KUKA KRL program: MyProgram_175().src

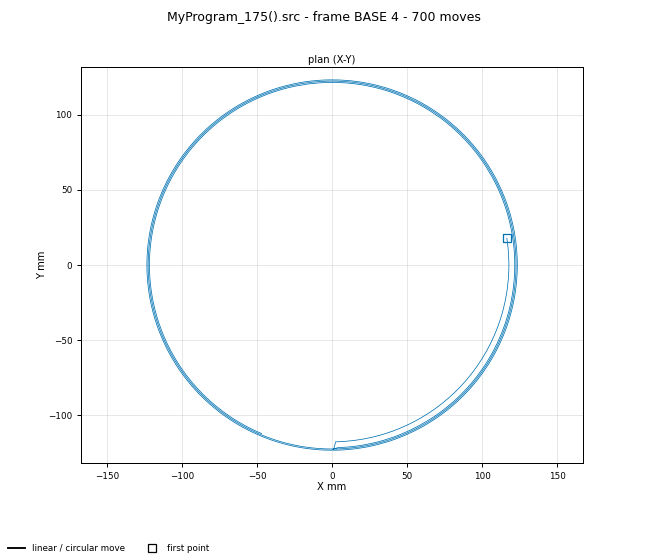
[picture p0: tool path of MyProgram_175().src in frame BASE 4, 700 of 700 moves have a stored position in this frame; points joined in program order, loops and branches not executed]
&ACCESS RVP
&REL 1
&PARAM TEMPLATE = C:\KRC\Roboter\Template\vorgabe
&PARAM EDITMASK = *
DEF MyProgram_175()
; ---- Setting reference (Base) ----
$BASE = BASE_DATA[4]

; --------------------------
; ---- Setting tool (TCP) ----
$TOOL = TOOL_DATA[3]
; --------------------------

$VEL.CP = VEL_APROX_PRINT
Startdeposition()
$VEL.CP = VEL_PRINT
LIN {X 116.3937,Y 17.9256,Z 129,A 4.4321,B 24.9467,C -1.6867,E1 25.1581,E2 441.6047} C_DIS
LIN {X 116.7972,Y 15.0743,Z 129,A 3.0217,B 24.947,C -1.6817,E1 25.1586,E2 443.0185} C_DIS
LIN {X 117.1569,Y 11.9651,Z 129,A 1.4665,B 24.9474,C -1.6752,E1 25.1591,E2 444.5798} C_DIS
LIN {X 117.4486,Y 8.67,Z 129,A -0.1015,B 24.9476,C -1.672,E1 25.1594,E2 446.1462} C_DIS
LIN {X 117.6272,Y 5.7574,Z 129,A -1.4975,B 24.9478,C -1.6685,E1 25.1596,E2 447.5421} C_DIS
LIN {X 117.7329,Y 2.8788,Z 129,A -2.8893,B 24.9481,C -1.6644,E1 25.1598,E2 448.9353} C_DIS
LIN {X 117.7651,Y -0.5226,Z 129,A -4.5792,B 24.9485,C -1.6573,E1 25.1598,E2 450.6318} C_DIS
LIN {X 117.7122,Y -3.559,Z 129,A -6.025,B 24.9487,C -1.654,E1 25.1597,E2 452.0768} C_DIS
LIN {X 117.5839,Y -6.5462,Z 129,A -7.4486,B 24.9489,C -1.6507,E1 25.1595,E2 453.4997} C_DIS
LIN {X 117.394,Y -9.3527,Z 129,A -8.8238,B 24.9492,C -1.6459,E1 25.1592,E2 454.8781} C_DIS
LIN {X 117.1208,Y -12.3096,Z 129,A -10.2202,B 24.9494,C -1.6435,E1 25.1588,E2 456.2718} C_DIS
LIN {X 116.796,Y -15.0832,Z 129,A -11.6081,B 24.9497,C -1.6377,E1 25.1583,E2 457.6654} C_DIS
LIN {X 116.3879,Y -17.9631,Z 129,A -13.0134,B 24.95,C -1.6335,E1 25.1578,E2 459.0722} C_DIS
LIN {X 115.8974,Y -20.8952,Z 129,A -14.4115,B 24.9501,C -1.6311,E1 25.1571,E2 460.4677} C_DIS
LIN {X 115.3444,Y -23.759,Z 129,A -15.8145,B 24.9504,C -1.6273,E1 25.1563,E2 461.8716} C_DIS
LIN {X 114.7348,Y -26.5469,Z 129,A -17.1994,B 24.9506,C -1.623,E1 25.1555,E2 463.2586} C_DIS
LIN {X 114.0503,Y -29.3488,Z 129,A -18.6126,B 24.9509,C -1.6179,E1 25.1545,E2 464.6755} C_DIS
LIN {X 113.3216,Y -32.0474,Z 129,A -20.0108,B 24.9513,C -1.6117,E1 25.1535,E2 466.0803} C_DIS
LIN {X 112.2615,Y -35.59,Z 129,A -21.7488,B 24.9515,C -1.6089,E1 25.1521,E2 467.8151} C_DIS
LIN {X 111.3572,Y -38.326,Z 129,A -23.1413,B 24.9517,C -1.6049,E1 25.1508,E2 469.2092} C_DIS
LIN {X 110.3859,Y -41.0399,Z 129,A -24.5345,B 24.952,C -1.6009,E1 25.1495,E2 470.6039} C_DIS
LIN {X 109.1507,Y -44.2152,Z 129,A -26.2203,B 24.9524,C -1.5944,E1 25.1478,E2 472.2957} C_DIS
LIN {X 107.975,Y -47.013,Z 129,A -27.6487,B 24.9525,C -1.5922,E1 25.1462,E2 473.7217} C_DIS
LIN {X 106.7548,Y -49.7216,Z 129,A -29.0647,B 24.9527,C -1.5891,E1 25.1445,E2 475.1371} C_DIS
LIN {X 105.5449,Y -52.2407,Z 129,A -30.4738,B 24.9531,C -1.5826,E1 25.1428,E2 476.5539} C_DIS
LIN {X 104.167,Y -54.9368,Z 129,A -31.8799,B 24.9531,C -1.5814,E1 25.141,E2 477.9555} C_DIS
LIN {X 102.7942,Y -57.4645,Z 129,A -33.2704,B 24.9534,C -1.5777,E1 25.1391,E2 479.3475} C_DIS
LIN {X 101.4046,Y -59.8827,Z 129,A -34.6519,B 24.9537,C -1.5725,E1 25.1372,E2 480.7341} C_DIS
LIN {X 99.8534,Y -62.4349,Z 129,A -36.083,B 24.9539,C -1.5693,E1 25.1351,E2 482.1655} C_DIS
LIN {X 98.3422,Y -64.7891,Z 129,A -37.4354,B 24.9541,C -1.5658,E1 25.133,E2 483.5193} C_DIS
LIN {X 96.7259,Y -67.1783,Z 129,A -38.8304,B 24.9543,C -1.5623,E1 25.1308,E2 484.9158} C_DIS
LIN {X 95.0339,Y -69.5512,Z 129,A -40.2395,B 24.9545,C -1.5587,E1 25.1285,E2 486.3264} C_DIS
LIN {X 93.2787,Y -71.8881,Z 129,A -41.6535,B 24.9547,C -1.5552,E1 25.1261,E2 487.742} C_DIS
LIN {X 91.4909,Y -74.1501,Z 129,A -43.0481,B 24.9549,C -1.5518,E1 25.1237,E2 489.1381} C_DIS
LIN {X 89.6483,Y -76.3676,Z 129,A -44.4513,B 24.9551,C -1.5481,E1 25.1212,E2 490.5437} C_DIS
LIN {X 87.728,Y -78.566,Z 129,A -45.8549,B 24.9553,C -1.5452,E1 25.1186,E2 491.9479} C_DIS
LIN {X 85.7806,Y -80.6877,Z 129,A -47.2487,B 24.9555,C -1.5419,E1 25.1159,E2 493.3432} C_DIS
LIN {X 83.7811,Y -82.7619,Z 129,A -48.6429,B 24.9556,C -1.5388,E1 25.1132,E2 494.7389} C_DIS
LIN {X 81.7314,Y -84.7867,Z 129,A -50.0452,B 24.9558,C -1.5353,E1 25.1104,E2 496.1434} C_DIS
LIN {X 79.6064,Y -86.785,Z 129,A -51.4495,B 24.956,C -1.5326,E1 25.1075,E2 497.5483} C_DIS
LIN {X 77.4591,Y -88.7069,Z 129,A -52.8446,B 24.9562,C -1.5297,E1 25.1046,E2 498.9449} C_DIS
LIN {X 75.2647,Y -90.5761,Z 129,A -54.2403,B 24.9563,C -1.5268,E1 25.1016,E2 500.3421} C_DIS
LIN {X 73.0251,Y -92.3913,Z 129,A -55.6361,B 24.9565,C -1.524,E1 25.0986,E2 501.7393} C_DIS
LIN {X 70.7095,Y -94.1753,Z 129,A -57.0586,B 24.9567,C -1.5209,E1 25.0954,E2 503.1639} C_DIS
LIN {X 68.3563,Y -95.897,Z 129,A -58.4643,B 24.9567,C -1.5185,E1 25.0922,E2 504.5702} C_DIS
LIN {X 65.9875,Y -97.5422,Z 129,A -59.8614,B 24.9569,C -1.516,E1 25.089,E2 505.9686} C_DIS
LIN {X 63.6275,Y -99.0977,Z 129,A -61.2294,B 24.9571,C -1.5136,E1 25.0858,E2 507.3377} C_DIS
LIN {X 61.1156,Y -100.6663,Z 129,A -62.6648,B 24.9572,C -1.5111,E1 25.0824,E2 508.7746} C_DIS
LIN {X 58.6405,Y -102.1279,Z 129,A -64.0379,B 24.9573,C -1.5097,E1 25.0791,E2 510.1468} C_DIS
LIN {X 56.131,Y -103.5284,Z 129,A -65.4376,B 24.9574,C -1.5071,E1 25.0756,E2 511.5484} C_DIS
LIN {X 53.4791,Y -104.9229,Z 129,A -66.8953,B 24.9576,C -1.5046,E1 25.072,E2 513.008} C_DIS
LIN {X 50.9395,Y -106.1791,Z 129,A -68.2585,B 24.9576,C -1.5031,E1 25.0686,E2 514.3712} C_DIS
LIN {X 48.3281,Y -107.3928,Z 129,A -69.6738,B 24.9578,C -1.5002,E1 25.065,E2 515.7897} C_DIS
LIN {X 45.6867,Y -108.5428,Z 129,A -71.0517,B 24.9578,C -1.4992,E1 25.0615,E2 517.1667} C_DIS
LIN {X 43.0999,Y -109.5957,Z 129,A -72.4452,B 24.9581,C -1.4956,E1 25.0578,E2 518.5655} C_DIS
LIN {X 40.3227,Y -110.6476,Z 129,A -73.8663,B 24.9581,C -1.4948,E1 25.0541,E2 519.9856} C_DIS
LIN {X 37.6045,Y -111.6007,Z 129,A -75.2508,B 24.9581,C -1.4938,E1 25.0505,E2 521.3698} C_DIS
LIN {X 34.8327,Y -112.4967,Z 129,A -76.7077,B 24.9584,C -1.4902,E1 25.0466,E2 522.8324} C_DIS
LIN {X 31.3934,Y -113.5067,Z 129,A -78.4167,B 24.9584,C -1.4898,E1 25.042,E2 524.5395} C_DIS
LIN {X 28.6049,Y -114.2414,Z 129,A -79.8167,B 24.9584,C -1.4885,E1 25.0382,E2 525.9405} C_DIS
LIN {X 25.7987,Y -114.9076,Z 129,A -81.2172,B 24.9586,C -1.4873,E1 25.0344,E2 527.342} C_DIS
LIN {X 22.9256,Y -115.5149,Z 129,A -82.6405,B 24.9586,C -1.4863,E1 25.0305,E2 528.7659} C_DIS
LIN {X 20.1009,Y -116.0398,Z 129,A -84.0367,B 24.9586,C -1.4852,E1 25.0267,E2 530.163} C_DIS
LIN {X 17.2609,Y -116.4962,Z 129,A -85.4392,B 24.9587,C -1.484,E1 25.0228,E2 531.567} C_DIS
LIN {X 14.409,Y -116.8833,Z 129,A -86.8328,B 24.9587,C -1.4834,E1 25.0189,E2 532.9609} C_DIS
LIN {X 11.5196,Y -117.2033,Z 129,A -88.2452,B 24.9588,C -1.4827,E1 25.015,E2 534.374} C_DIS
LIN {X 8.653,Y -117.4498,Z 129,A -89.7448,B 24.9591,C -1.4775,E1 25.0108,E2 535.8853} C_DIS
LIN {X 5.7539,Y -117.6274,Z 129,A -91.0554,B 24.9589,C -1.4815,E1 25.0072,E2 537.1858} C_DIS
LIN {X 2.394,Y -117.7418,Z 129,A -92.7403,B 24.959,C -1.4788,E1 25.0024,E2 538.8768} C_DIS
LIN {X 2.394,Y -117.7418,Z 129,A -92.7403,B 24.959,C -1.4788,E1 25.0024,E2 538.8768} C_DIS
Enddeposition()
LIN {X 0.876,Y -123.3662,Z 130,A -92.9891,B 24.9627,C -1.4112,E1 25.0013,E2 539.2857} C_DIS
Startdeposition()
$VEL.CP = VEL_PRINT
LIN {X 3.429,Y -123.3221,Z 130,A -91.439,B 24.9617,C -1.4291,E1 25.0058,E2 537.6935} C_DIS
LIN {X 6.0536,Y -123.2229,Z 130,A -90.0878,B 24.9614,C -1.4359,E1 25.0096,E2 536.3266} C_DIS
LIN {X 9.4299,Y -123.0089,Z 130,A -88.6359,B 24.9616,C -1.4309,E1 25.0136,E2 534.8873} C_DIS
LIN {X 12.4918,Y -122.7357,Z 130,A -87.2244,B 24.9616,C -1.4309,E1 25.0175,E2 533.4767} C_DIS
LIN {X 15.102,Y -122.4437,Z 130,A -86.0061,B 24.9616,C -1.4315,E1 25.0209,E2 532.2577} C_DIS
LIN {X 18.4991,Y -121.9749,Z 130,A -84.4157,B 24.9616,C -1.4325,E1 25.0253,E2 530.6664} C_DIS
LIN {X 21.0918,Y -121.5552,Z 130,A -83.0658,B 24.9612,C -1.4398,E1 25.029,E2 529.3006} C_DIS
LIN {X 24.0686,Y -121.001,Z 130,A -81.6622,B 24.9612,C -1.4409,E1 25.0329,E2 527.8961} C_DIS
LIN {X 27.422,Y -120.2835,Z 130,A -80.2048,B 24.9614,C -1.4358,E1 25.0368,E2 526.4527} C_DIS
LIN {X 29.9768,Y -119.6742,Z 130,A -78.9876,B 24.9614,C -1.4368,E1 25.0401,E2 525.2348} C_DIS
LIN {X 33.291,Y -118.7931,Z 130,A -77.5658,B 24.9617,C -1.4302,E1 25.0439,E2 523.831} C_DIS
LIN {X 35.8129,Y -118.0592,Z 130,A -76.1817,B 24.9612,C -1.4397,E1 25.0477,E2 522.4269} C_DIS
LIN {X 38.6994,Y -117.1447,Z 130,A -74.7791,B 24.9611,C -1.4412,E1 25.0514,E2 521.0233} C_DIS
LIN {X 41.5626,Y -116.1597,Z 130,A -73.3767,B 24.9611,C -1.4429,E1 25.0551,E2 519.6198} C_DIS
LIN {X 44.7745,Y -114.958,Z 130,A -71.784,B 24.9609,C -1.4451,E1 25.0592,E2 518.0252} C_DIS
LIN {X 47.2122,Y -113.9804,Z 130,A -70.5726,B 24.9609,C -1.4464,E1 25.0624,E2 516.8135} C_DIS
LIN {X 50.3612,Y -112.6225,Z 130,A -68.9852,B 24.9607,C -1.4486,E1 25.0664,E2 515.2248} C_DIS
LIN {X 53.11,Y -111.3527,Z 130,A -67.7507,B 24.961,C -1.4424,E1 25.0695,E2 514.0082} C_DIS
LIN {X 55.4692,Y -110.1985,Z 130,A -66.2126,B 24.9601,C -1.4602,E1 25.0735,E2 512.4322} C_DIS
LIN {X 58.5098,Y -108.6126,Z 130,A -64.7813,B 24.9603,C -1.455,E1 25.0769,E2 511.0173} C_DIS
LIN {X 61.1577,Y -107.144,Z 130,A -63.5474,B 24.9607,C -1.4489,E1 25.0799,E2 509.8014} C_DIS
LIN {X 63.7687,Y -105.6108,Z 130,A -62.0577,B 24.9603,C -1.4557,E1 25.0835,E2 508.3002} C_DIS
LIN {X 66.3413,Y -104.014,Z 130,A -60.5698,B 24.9599,C -1.4625,E1 25.0871,E2 506.8009} C_DIS
LIN {X 68.601,Y -102.5394,Z 130,A -59.3612,B 24.9599,C -1.4628,E1 25.0899,E2 505.5958} C_DIS
LIN {X 71.0383,Y -100.8667,Z 130,A -57.9646,B 24.9597,C -1.4668,E1 25.0931,E2 504.1945} C_DIS
LIN {X 73.8133,Y -98.8518,Z 130,A -56.3792,B 24.9595,C -1.4698,E1 25.0966,E2 502.6075} C_DIS
LIN {X 75.9021,Y -97.2595,Z 130,A -55.0333,B 24.959,C -1.4788,E1 25.0997,E2 501.2453} C_DIS
LIN {X 78.2661,Y -95.3675,Z 130,A -53.6536,B 24.959,C -1.4806,E1 25.1026,E2 499.8665} C_DIS
LIN {X 80.5829,Y -93.418,Z 130,A -52.2344,B 24.9587,C -1.4845,E1 25.1057,E2 498.4437} C_DIS
LIN {X 83.1471,Y -91.1409,Z 130,A -50.9478,B 24.9594,C -1.4729,E1 25.1083,E2 497.1898} C_DIS
LIN {X 85.0697,Y -89.3515,Z 130,A -49.4363,B 24.9584,C -1.4905,E1 25.1114,E2 495.6428} C_DIS
LIN {X 87.2368,Y -87.2368,Z 130,A -48.0373,B 24.9582,C -1.4936,E1 25.1142,E2 494.2424} C_DIS
LIN {X 89.6265,Y -84.7772,Z 130,A -46.7511,B 24.9588,C -1.4822,E1 25.1166,E2 492.9888} C_DIS
LIN {X 91.4123,Y -82.8513,Z 130,A -45.2399,B 24.9578,C -1.5001,E1 25.1195,E2 491.4421} C_DIS
LIN {X 93.6784,Y -80.2773,Z 130,A -43.7876,B 24.958,C -1.4971,E1 25.1222,E2 490.0032} C_DIS
LIN {X 95.3675,Y -78.2661,Z 130,A -42.443,B 24.9575,C -1.5067,E1 25.1246,E2 488.6423} C_DIS
LIN {X 97.2595,Y -75.9021,Z 130,A -41.1765,B 24.9577,C -1.5034,E1 25.1267,E2 487.3895} C_DIS
LIN {X 99.3301,Y -73.1684,Z 130,A -39.5931,B 24.9574,C -1.5074,E1 25.1294,E2 485.8044} C_DIS
LIN {X 101.0958,Y -70.7087,Z 130,A -38.1953,B 24.9572,C -1.5109,E1 25.1316,E2 484.4051} C_DIS
LIN {X 102.8755,Y -68.0929,Z 130,A -36.9573,B 24.9577,C -1.5033,E1 25.1335,E2 483.191} C_DIS
LIN {X 104.4436,Y -65.663,Z 130,A -35.5665,B 24.9573,C -1.5096,E1 25.1357,E2 481.7924} C_DIS
LIN {X 106.0236,Y -63.0801,Z 130,A -34.1685,B 24.9571,C -1.5132,E1 25.1377,E2 480.3929} C_DIS
LIN {X 107.344,Y -60.8096,Z 130,A -32.79,B 24.9564,C -1.5249,E1 25.1396,E2 478.994} C_DIS
LIN {X 108.991,Y -57.8017,Z 130,A -31.2074,B 24.9562,C -1.5292,E1 25.1417,E2 477.4096} C_DIS
LIN {X 110.3767,Y -55.1096,Z 130,A -29.9764,B 24.9565,C -1.5245,E1 25.1433,E2 476.1962} C_DIS
LIN {X 111.5265,Y -52.7481,Z 130,A -28.5983,B 24.9558,C -1.5363,E1 25.1449,E2 474.7977} C_DIS
LIN {X 112.9479,Y -49.6272,Z 130,A -27.0159,B 24.9555,C -1.5407,E1 25.1468,E2 473.2135} C_DIS
LIN {X 113.9804,Y -47.2122,Z 130,A -25.8038,B 24.9553,C -1.5441,E1 25.1481,E2 472.0002} C_DIS
LIN {X 115.2469,Y -44.0254,Z 130,A -24.177,B 24.9549,C -1.5509,E1 25.1497,E2 470.3665} C_DIS
LIN {X 116.2927,Y -41.1838,Z 130,A -22.825,B 24.9549,C -1.5525,E1 25.151,E2 469.0181} C_DIS
LIN {X 117.2683,Y -38.3174,Z 130,A -21.4284,B 24.9546,C -1.5565,E1 25.1522,E2 467.62} C_DIS
LIN {X 118.1734,Y -35.428,Z 130,A -20.1978,B 24.9549,C -1.552,E1 25.1532,E2 466.407} C_DIS
LIN {X 119.0072,Y -32.5172,Z 130,A -18.6351,B 24.9541,C -1.5645,E1 25.1544,E2 464.8237} C_DIS
LIN {X 119.6742,Y -29.9768,Z 130,A -17.3374,B 24.9537,C -1.5724,E1 25.1553,E2 463.5149} C_DIS
LIN {X 120.4667,Y -26.6053,Z 130,A -15.8289,B 24.9537,C -1.5726,E1 25.1563,E2 462.0148} C_DIS
LIN {X 121.001,Y -24.0686,Z 130,A -14.4988,B 24.9531,C -1.5829,E1 25.157,E2 460.6681} C_DIS
LIN {X 121.5552,Y -21.0918,Z 130,A -13.2337,B 24.9532,C -1.5803,E1 25.1576,E2 459.4166} C_DIS
LIN {X 122.0927,Y -17.7049,Z 130,A -11.6521,B 24.9529,C -1.5849,E1 25.1583,E2 457.8334} C_DIS
LIN {X 122.6198,Y -13.5983,Z 130,A -9.7423,B 24.9526,C -1.5905,E1 25.1589,E2 455.9216} C_DIS
LIN {X 122.9486,Y -10.1848,Z 130,A -8.3272,B 24.9528,C -1.5867,E1 25.1593,E2 454.5239} C_DIS
LIN {X 123.1615,Y -7.1644,Z 130,A -6.9306,B 24.9526,C -1.5908,E1 25.1596,E2 453.1259} C_DIS
LIN {X 123.2879,Y -4.541,Z 130,A -5.4214,B 24.9515,C -1.6097,E1 25.1597,E2 451.5813} C_DIS
LIN {X 123.3622,Y -1.514,Z 130,A -4.0379,B 24.9512,C -1.6131,E1 25.1597,E2 450.198} C_DIS
LIN {X 123.3607,Y 1.5958,Z 130,A -2.6187,B 24.951,C -1.6165,E1 25.1597,E2 448.779} C_DIS
LIN {X 123.2707,Y 4.942,Z 130,A -1.3446,B 24.9516,C -1.6073,E1 25.1597,E2 447.5344} C_DIS
LIN {X 123.1123,Y 7.9658,Z 130,A 0.0521,B 24.9513,C -1.6114,E1 25.1594,E2 446.1363} C_DIS
LIN {X 122.9166,Y 10.5849,Z 130,A 1.5614,B 24.9502,C -1.6301,E1 25.1591,E2 444.5918} C_DIS
LIN {X 122.5731,Y 13.997,Z 130,A 3.0115,B 24.9503,C -1.628,E1 25.1586,E2 443.1553} C_DIS
LIN {X 122.1927,Y 17.0009,Z 130,A 4.4082,B 24.9501,C -1.632,E1 25.1581,E2 441.7573} C_DIS
LIN {X 121.7387,Y 19.9945,Z 130,A 5.6386,B 24.9504,C -1.6276,E1 25.1576,E2 440.5446} C_DIS
LIN {X 121.2113,Y 22.9761,Z 130,A 7.2015,B 24.9496,C -1.64,E1 25.1568,E2 438.9615} C_DIS
LIN {X 120.611,Y 25.9439,Z 130,A 8.6253,B 24.9493,C -1.6454,E1 25.156,E2 437.5334} C_DIS
LIN {X 119.6742,Y 29.9768,Z 130,A 10.5089,B 24.949,C -1.6494,E1 25.1548,E2 435.6512} C_DIS
LIN {X 118.9025,Y 32.9048,Z 130,A 11.9058,B 24.9488,C -1.6533,E1 25.1537,E2 434.2532} C_DIS
LIN {X 118.0592,Y 35.8129,Z 130,A 13.3029,B 24.9485,C -1.6572,E1 25.1526,E2 432.855} C_DIS
LIN {X 117.1448,Y 38.6994,Z 130,A 14.8315,B 24.9479,C -1.6677,E1 25.1513,E2 431.3101} C_DIS
LIN {X 116.1597,Y 41.5626,Z 130,A 16.0973,B 24.9481,C -1.6648,E1 25.1501,E2 430.0584} C_DIS
LIN {X 115.1048,Y 44.4008,Z 130,A 17.5072,B 24.9478,C -1.6692,E1 25.1487,E2 428.6459} C_DIS
LIN {X 113.8245,Y 47.5822,Z 130,A 18.911,B 24.9481,C -1.6643,E1 25.1473,E2 427.2613} C_DIS
LIN {X 112.7875,Y 49.9952,Z 130,A 20.3887,B 24.9471,C -1.6809,E1 25.1456,E2 425.7526} C_DIS
LIN {X 111.3527,Y 53.11,Z 130,A 21.7062,B 24.9476,C -1.6716,E1 25.1441,E2 424.4641} C_DIS
LIN {X 110.1985,Y 55.4692,Z 130,A 23.0851,B 24.9469,C -1.6831,E1 25.1423,E2 423.0655} C_DIS
LIN {X 108.6126,Y 58.5098,Z 130,A 24.6684,B 24.9467,C -1.6871,E1 25.1403,E2 421.4811} C_DIS
LIN {X 107.144,Y 61.1577,Z 130,A 26.0664,B 24.9464,C -1.6906,E1 25.1383,E2 420.0822} C_DIS
LIN {X 105.6108,Y 63.7687,Z 130,A 27.2981,B 24.9468,C -1.6856,E1 25.1366,E2 418.8686} C_DIS
LIN {X 104.2309,Y 66.0035,Z 130,A 28.7053,B 24.946,C -1.6982,E1 25.1345,E2 417.4386} C_DIS
LIN {X 102.3546,Y 68.874,Z 130,A 30.0946,B 24.9463,C -1.6922,E1 25.1324,E2 416.0704} C_DIS
LIN {X 100.6335,Y 71.3651,Z 130,A 31.6599,B 24.9456,C -1.7038,E1 25.1299,E2 414.4854} C_DIS
LIN {X 98.8518,Y 73.8133,Z 130,A 33.0587,B 24.9454,C -1.707,E1 25.1275,E2 413.0859} C_DIS
LIN {X 97.0106,Y 76.217,Z 130,A 34.2907,B 24.9457,C -1.7017,E1 25.1255,E2 411.8721} C_DIS
LIN {X 95.1109,Y 78.5748,Z 130,A 35.6897,B 24.9455,C -1.7047,E1 25.123,E2 410.4725} C_DIS
LIN {X 93.418,Y 80.5829,Z 130,A 37.0705,B 24.9448,C -1.7156,E1 25.1205,E2 409.0724} C_DIS
LIN {X 91.4123,Y 82.8513,Z 130,A 38.4701,B 24.9447,C -1.7185,E1 25.1179,E2 407.6721} C_DIS
LIN {X 89.0729,Y 85.3587,Z 130,A 39.888,B 24.945,C -1.7134,E1 25.1152,E2 406.2724} C_DIS
LIN {X 86.9512,Y 87.519,Z 130,A 41.4546,B 24.9443,C -1.7245,E1 25.1121,E2 404.6864} C_DIS
LIN {X 84.7772,Y 89.6265,Z 130,A 42.6878,B 24.9446,C -1.7189,E1 25.1096,E2 403.4715} C_DIS
LIN {X 82.8513,Y 91.4123,Z 130,A 44.0692,B 24.944,C -1.7294,E1 25.1067,E2 402.071} C_DIS
LIN {X 80.3955,Y 93.5777,Z 130,A 45.5306,B 24.944,C -1.7295,E1 25.1037,E2 400.615} C_DIS
LIN {X 78.2661,Y 95.3675,Z 130,A 46.87,B 24.9436,C -1.7343,E1 25.1008,E2 399.2693} C_DIS
LIN {X 75.5841,Y 97.5045,Z 130,A 48.4562,B 24.9435,C -1.737,E1 25.0973,E2 397.6826} C_DIS
LIN {X 73.1684,Y 99.3301,Z 130,A 49.6903,B 24.9438,C -1.7311,E1 25.0946,E2 396.467} C_DIS
LIN {X 71.0383,Y 100.8667,Z 130,A 51.2044,B 24.9428,C -1.7477,E1 25.0911,E2 394.919} C_DIS
LIN {X 68.2064,Y 102.8007,Z 130,A 52.6595,B 24.943,C -1.7436,E1 25.0877,E2 393.4785} C_DIS
LIN {X 66.0035,Y 104.2309,Z 130,A 54.0337,B 24.9424,C -1.7531,E1 25.0844,E2 392.0863} C_DIS
LIN {X 63.0801,Y 106.0236,Z 130,A 55.2956,B 24.9433,C -1.7393,E1 25.0815,E2 390.8609} C_DIS
LIN {X 60.8096,Y 107.344,Z 130,A 56.8108,B 24.9422,C -1.7555,E1 25.0778,E2 389.312} C_DIS
LIN {X 57.8017,Y 108.991,Z 130,A 58.0995,B 24.9431,C -1.7429,E1 25.0747,E2 388.0567} C_DIS
LIN {X 55.1096,Y 110.3767,Z 130,A 59.6689,B 24.9424,C -1.7527,E1 25.0707,E2 386.4685} C_DIS
LIN {X 52.3842,Y 111.696,Z 130,A 60.9044,B 24.9429,C -1.7461,E1 25.0676,E2 385.2518} C_DIS
LIN {X 49.9952,Y 112.7875,Z 130,A 62.2885,B 24.9422,C -1.7555,E1 25.0641,E2 383.8489} C_DIS
LIN {X 47.2122,Y 113.9804,Z 130,A 63.6918,B 24.9422,C -1.7568,E1 25.0605,E2 382.4457} C_DIS
LIN {X 44.4008,Y 115.1048,Z 130,A 65.0947,B 24.9421,C -1.7581,E1 25.0568,E2 381.0429} C_DIS
LIN {X 41.5081,Y 116.1789,Z 130,A 66.5008,B 24.9421,C -1.7581,E1 25.0531,E2 379.6396} C_DIS
LIN {X 38.6994,Y 117.1447,Z 130,A 67.9019,B 24.9419,C -1.7604,E1 25.0494,E2 378.236} C_DIS
LIN {X 35.428,Y 118.1734,Z 130,A 69.4918,B 24.9419,C -1.7615,E1 25.0452,E2 376.6463} C_DIS
LIN {X 32.5172,Y 119.0072,Z 130,A 70.7285,B 24.9423,C -1.7543,E1 25.0419,E2 375.4285} C_DIS
LIN {X 29.9768,Y 119.6742,Z 130,A 72.2466,B 24.9413,C -1.7694,E1 25.0377,E2 373.8771} C_DIS
LIN {X 27.0309,Y 120.3739,Z 130,A 73.6515,B 24.9413,C -1.7701,E1 25.0339,E2 372.4726} C_DIS
LIN {X 24.0686,Y 121.001,Z 130,A 75.0932,B 24.9411,C -1.7724,E1 25.0299,E2 371.027} C_DIS
LIN {X 19.5986,Y 121.8049,Z 130,A 77.164,B 24.9411,C -1.7713,E1 25.0242,E2 368.961} C_DIS
LIN {X 16.2053,Y 122.3008,Z 130,A 78.4557,B 24.9421,C -1.7574,E1 25.0208,E2 367.7033} C_DIS
LIN {X 13.5983,Y 122.6198,Z 130,A 79.8428,B 24.9416,C -1.7656,E1 25.0169,E2 366.298} C_DIS
LIN {X 10.1848,Y 122.9486,Z 130,A 81.2672,B 24.9421,C -1.7578,E1 25.013,E2 364.8928} C_DIS
LIN {X 7.1644,Y 123.1615,Z 130,A 82.6735,B 24.9421,C -1.7578,E1 25.009,E2 363.4871} C_DIS
LIN {X 4.541,Y 123.2879,Z 130,A 84.1939,B 24.9412,C -1.7719,E1 25.0047,E2 361.9337} C_DIS
LIN {X 1.1125,Y 123.3647,Z 130,A 85.4866,B 24.9421,C -1.7576,E1 25.0012,E2 360.6752} C_DIS
LIN {X -1.514,Y 123.3622,Z 130,A 87.0075,B 24.9412,C -1.7714,E1 24.9969,E2 359.1214} C_DIS
LIN {X -4.942,Y 123.2707,Z 130,A 88.3006,B 24.9421,C -1.7569,E1 24.9933,E2 357.8625} C_DIS
LIN {X -7.9658,Y 123.1123,Z 130,A 89.7082,B 24.9421,C -1.7564,E1 24.9894,E2 356.4557} C_DIS
LIN {X -10.9847,Y 122.8797,Z 130,A 91.2835,B 24.9417,C -1.7637,E1 24.985,E2 354.8624} C_DIS
LIN {X -13.8703,Y 122.588,Z 130,A 92.5176,B 24.9421,C -1.7577,E1 24.9816,E2 353.6418} C_DIS
LIN {X -16.6034,Y 122.2492,Z 130,A 94.0457,B 24.9414,C -1.7685,E1 24.9773,E2 352.087} C_DIS
LIN {X -19.9945,Y 121.7387,Z 130,A 95.34,B 24.9424,C -1.7535,E1 24.9738,E2 350.8271} C_DIS
LIN {X -22.9761,Y 121.2113,Z 130,A 96.8258,B 24.9422,C -1.7561,E1 24.9697,E2 349.3335} C_DIS
LIN {X -25.9439,Y 120.611,Z 130,A 98.3448,B 24.9419,C -1.7601,E1 24.9655,E2 347.8033} C_DIS
LIN {X -28.9432,Y 119.9264,Z 130,A 99.569,B 24.9426,C -1.7493,E1 24.9623,E2 346.603} C_DIS
LIN {X -31.4432,Y 119.2974,Z 130,A 101.0899,B 24.9417,C -1.7631,E1 24.9581,E2 345.0474} C_DIS
LIN {X -34.3614,Y 118.4898,Z 130,A 102.3665,B 24.9422,C -1.7555,E1 24.9547,E2 343.7866} C_DIS
LIN {X -37.2589,Y 117.6108,Z 130,A 103.7764,B 24.9423,C -1.7541,E1 24.9509,E2 342.3776} C_DIS
LIN {X -40.134,Y 116.661,Z 130,A 105.1862,B 24.9424,C -1.7525,E1 24.9472,E2 340.969} C_DIS
LIN {X -42.9849,Y 115.641,Z 130,A 106.7293,B 24.9421,C -1.757,E1 24.9431,E2 339.4122} C_DIS
LIN {X -46.1818,Y 114.3999,Z 130,A 108.1935,B 24.9427,C -1.7489,E1 24.9393,E2 337.9639} C_DIS
LIN {X -48.7024,Y 113.3511,Z 130,A 109.5628,B 24.9425,C -1.7517,E1 24.9358,E2 336.5848} C_DIS
LIN {X -51.7395,Y 111.996,Z 130,A 111.0152,B 24.9429,C -1.7451,E1 24.9321,E2 335.1444} C_DIS
LIN {X -54.1128,Y 110.8708,Z 130,A 112.2392,B 24.943,C -1.7433,E1 24.9291,E2 333.9216} C_DIS
LIN {X -56.8174,Y 109.5095,Z 130,A 113.6506,B 24.9432,C -1.7412,E1 24.9256,E2 332.5114} C_DIS
LIN {X -59.8383,Y 107.8864,Z 130,A 115.2491,B 24.9433,C -1.7387,E1 24.9216,E2 330.9143} C_DIS
LIN {X -62.1223,Y 106.5897,Z 130,A 116.6066,B 24.9431,C -1.7428,E1 24.9183,E2 329.5431} C_DIS
LIN {X -64.7194,Y 105.033,Z 130,A 118.0188,B 24.9432,C -1.7404,E1 24.915,E2 328.1322} C_DIS
LIN {X -67.2776,Y 103.4131,Z 130,A 119.2975,B 24.9438,C -1.7319,E1 24.912,E2 326.8696} C_DIS
LIN {X -70.1248,Y 101.5017,Z 130,A 120.8971,B 24.944,C -1.729,E1 24.9083,E2 325.2714} C_DIS
LIN {X -72.2708,Y 99.9873,Z 130,A 122.2553,B 24.9437,C -1.7327,E1 24.9052,E2 323.8996} C_DIS
LIN {X -74.7028,Y 98.1836,Z 130,A 123.6683,B 24.9439,C -1.73,E1 24.9021,E2 322.488} C_DIS
LIN {X -77.4018,Y 96.068,Z 130,A 124.9666,B 24.945,C -1.7133,E1 24.8993,E2 321.2246} C_DIS
LIN {X -79.7361,Y 94.1395,Z 130,A 126.3794,B 24.9452,C -1.7105,E1 24.8963,E2 319.8132} C_DIS
LIN {X -81.7233,Y 92.4221,Z 130,A 127.9073,B 24.9445,C -1.7215,E1 24.893,E2 318.2531} C_DIS
LIN {X -83.9668,Y 90.3887,Z 130,A 129.1875,B 24.945,C -1.7125,E1 24.8904,E2 316.9892} C_DIS
LIN {X -86.4454,Y 88.0187,Z 130,A 130.6198,B 24.9457,C -1.7015,E1 24.8876,E2 315.577} C_DIS
LIN {X -88.4404,Y 86.0149,Z 130,A 132.024,B 24.9457,C -1.7023,E1 24.8848,E2 314.165} C_DIS
LIN {X -90.6601,Y 83.671,Z 130,A 133.6159,B 24.9457,C -1.7027,E1 24.8817,E2 312.5653} C_DIS
LIN {X -92.6862,Y 81.4209,Z 130,A 135.0299,B 24.9459,C -1.6994,E1 24.8791,E2 311.1527} C_DIS
LIN {X -94.3999,Y 79.4305,Z 130,A 136.2566,B 24.9461,C -1.6965,E1 24.8769,E2 309.9273} C_DIS
LIN {X -96.5697,Y 76.7749,Z 130,A 137.6895,B 24.9468,C -1.6851,E1 24.8744,E2 308.5147} C_DIS
LIN {X -98.1836,Y 74.7028,Z 130,A 139.0852,B 24.9465,C -1.6896,E1 24.872,E2 307.1017} C_DIS
LIN {X -99.9873,Y 72.2708,Z 130,A 140.4998,B 24.9467,C -1.6861,E1 24.8697,E2 305.6887} C_DIS
LIN {X -101.7308,Y 69.7952,Z 130,A 142.0478,B 24.9466,C -1.6885,E1 24.8672,E2 304.1274} C_DIS
LIN {X -103.6942,Y 66.8396,Z 130,A 143.537,B 24.9473,C -1.6768,E1 24.8649,E2 302.6586} C_DIS
LIN {X -105.2415,Y 64.3764,Z 130,A 144.9317,B 24.9474,C -1.6748,E1 24.8629,E2 301.2614} C_DIS
LIN {X -106.7897,Y 61.7742,Z 130,A 146.178,B 24.9481,C -1.6636,E1 24.8612,E2 300.0352} C_DIS
LIN {X -108.2735,Y 59.1349,Z 130,A 147.762,B 24.9479,C -1.6673,E1 24.859,E2 298.4341} C_DIS
LIN {X -110.1985,Y 55.4692,Z 130,A 149.7664,B 24.948,C -1.6651,E1 24.8564,E2 296.4243} C_DIS
LIN {X -111.696,Y 52.3842,Z 130,A 151.1316,B 24.949,C -1.6503,E1 24.8548,E2 295.0871} C_DIS
LIN {X -112.7875,Y 49.9952,Z 130,A 152.5284,B 24.9487,C -1.6543,E1 24.8532,E2 293.673} C_DIS
LIN {X -114.1318,Y 46.8404,Z 130,A 154.1316,B 24.949,C -1.6499,E1 24.8514,E2 292.0714} C_DIS
LIN {X -115.1048,Y 44.4008,Z 130,A 155.4169,B 24.949,C -1.6489,E1 24.8501,E2 290.7812} C_DIS
LIN {X -116.1597,Y 41.5626,Z 130,A 156.9088,B 24.949,C -1.6483,E1 24.8487,E2 289.2824} C_DIS
LIN {X -117.2683,Y 38.3174,Z 130,A 158.21,B 24.9502,C -1.6304,E1 24.8476,E2 288.0163} C_DIS
LIN {X -118.1734,Y 35.428,Z 130,A 159.7947,B 24.95,C -1.6338,E1 24.8463,E2 286.4144} C_DIS
LIN {X -119.0072,Y 32.5172,Z 130,A 161.2106,B 24.9502,C -1.6297,E1 24.8452,E2 285.0001} C_DIS
LIN {X -119.7694,Y 29.5868,Z 130,A 162.6266,B 24.9505,C -1.6256,E1 24.8442,E2 283.5856} C_DIS
LIN {X -120.3739,Y 27.0309,Z 130,A 163.9885,B 24.9503,C -1.6279,E1 24.8434,E2 282.2102} C_DIS
LIN {X -121.001,Y 24.0686,Z 130,A 165.4044,B 24.9506,C -1.6238,E1 24.8426,E2 280.7959} C_DIS
LIN {X -121.5552,Y 21.0918,Z 130,A 166.687,B 24.9512,C -1.6137,E1 24.842,E2 279.5295} C_DIS
LIN {X -122.0927,Y 17.7049,Z 130,A 168.2907,B 24.9515,C -1.6091,E1 24.8413,E2 277.9274} C_DIS
LIN {X -122.6198,Y 13.5983,Z 130,A 170.2274,B 24.9518,C -1.6033,E1 24.8407,E2 275.9929} C_DIS
LIN {X -122.9486,Y 10.1848,Z 130,A 171.6621,B 24.9526,C -1.5912,E1 24.8403,E2 274.5784} C_DIS
LIN {X -123.1615,Y 7.1644,Z 130,A 173.0784,B 24.9528,C -1.587,E1 24.84,E2 273.1636} C_DIS
LIN {X -123.2879,Y 4.541,Z 130,A 174.6093,B 24.9522,C -1.5967,E1 24.8398,E2 271.6004} C_DIS
LIN {X -123.3622,Y 1.514,Z 130,A 176.0122,B 24.9525,C -1.5919,E1 24.8398,E2 270.2004} C_DIS
LIN {X -123.3622,Y -1.514,Z 130,A 177.4415,B 24.9527,C -1.5884,E1 24.8398,E2 268.771} C_DIS
LIN {X -123.2707,Y -4.942,Z 130,A 178.7429,B 24.9538,C -1.5704,E1 24.8399,E2 267.5047} C_DIS
LIN {X -123.1123,Y -7.9658,Z 130,A -179.6079,B 24.9534,C -1.5765,E1 24.8402,E2 265.831} C_DIS
LIN {X -122.8797,Y -10.9847,Z 130,A -178.2561,B 24.9538,C -1.5695,E1 24.8405,E2 264.4877} C_DIS
LIN {X -122.5731,Y -13.997,Z 130,A -177.009,B 24.9545,C -1.558,E1 24.8409,E2 263.2606} C_DIS
LIN {X -122.2492,Y -16.6034,Z 130,A -175.4784,B 24.9539,C -1.5678,E1 24.8415,E2 261.6975} C_DIS
LIN {X -121.7387,Y -19.9945,Z 130,A -174.0534,B 24.9547,C -1.5553,E1 24.8421,E2 260.2938} C_DIS
LIN {X -121.2113,Y -22.9761,Z 130,A -172.7614,B 24.9552,C -1.5458,E1 24.8427,E2 259.0168} C_DIS
LIN {X -120.611,Y -25.9439,Z 130,A -171.1766,B 24.955,C -1.5492,E1 24.8436,E2 257.4145} C_DIS
LIN {X -119.9379,Y -28.896,Z 130,A -169.7235,B 24.9552,C -1.5469,E1 24.8445,E2 255.9584} C_DIS
LIN {X -119.2974,Y -31.4432,Z 130,A -168.3995,B 24.9552,C -1.5477,E1 24.8455,E2 254.6248} C_DIS
LIN {X -118.4898,Y -34.3614,Z 130,A -167.1174,B 24.9557,C -1.5378,E1 24.8465,E2 253.3587} C_DIS
LIN {X -117.6108,Y -37.2589,Z 130,A -165.7016,B 24.9559,C -1.5339,E1 24.8476,E2 251.9441} C_DIS
LIN {X -116.661,Y -40.134,Z 130,A -164.2865,B 24.9561,C -1.5301,E1 24.8489,E2 250.5301} C_DIS
LIN {X -115.641,Y -42.9849,Z 130,A -162.7379,B 24.9561,C -1.5322,E1 24.8504,E2 248.9677} C_DIS
LIN {X -114.3999,Y -46.1818,Z 130,A -161.4373,B 24.957,C -1.5145,E1 24.8517,E2 247.7019} C_DIS
LIN {X -113.2741,Y -48.879,Z 130,A -159.8693,B 24.9567,C -1.5199,E1 24.8534,E2 246.1124} C_DIS
LIN {X -111.996,Y -51.7395,Z 130,A -158.4384,B 24.957,C -1.5146,E1 24.8551,E2 244.6862} C_DIS
LIN {X -110.8708,Y -54.1128,Z 130,A -157.2112,B 24.9572,C -1.5115,E1 24.8566,E2 243.4599} C_DIS
LIN {X -109.3694,Y -57.0833,Z 130,A -155.6242,B 24.9573,C -1.509,E1 24.8586,E2 241.8704} C_DIS
LIN {X -107.8864,Y -59.8383,Z 130,A -154.1943,B 24.9576,C -1.5039,E1 24.8605,E2 240.445} C_DIS
LIN {X -106.5897,Y -62.1223,Z 130,A -152.8342,B 24.9575,C -1.5069,E1 24.8624,E2 239.0707} C_DIS
LIN {X -104.7145,Y -65.2293,Z 130,A -151.3303,B 24.9582,C -1.4942,E1 24.8646,E2 237.5892} C_DIS
LIN {X -103.4131,Y -67.2776,Z 130,A -150.1389,B 24.9582,C -1.4942,E1 24.8664,E2 236.3921} C_DIS
LIN {X -101.7308,Y -69.7952,Z 130,A -148.7248,B 24.9584,C -1.4909,E1 24.8686,E2 234.9788} C_DIS
LIN {X -99.9873,Y -72.2708,Z 130,A -147.1779,B 24.9582,C -1.4937,E1 24.8711,E2 233.4176} C_DIS
LIN {X -97.9386,Y -75.0208,Z 130,A -145.6659,B 24.9586,C -1.4861,E1 24.8737,E2 231.9164} C_DIS
LIN {X -96.068,Y -77.4018,Z 130,A -144.4649,B 24.9593,C -1.4734,E1 24.8757,E2 230.74} C_DIS
LIN {X -94.3999,Y -79.4305,Z 130,A -143.0703,B 24.9591,C -1.4784,E1 24.8782,E2 229.327} C_DIS
LIN {X -92.1543,Y -82.0224,Z 130,A -141.4696,B 24.9592,C -1.4751,E1 24.8812,E2 227.727} C_DIS
LIN {X -90.3887,Y -83.9668,Z 130,A -140.2439,B 24.9594,C -1.4726,E1 24.8835,E2 226.5019} C_DIS
LIN {X -88.0187,Y -86.4454,Z 130,A -138.812,B 24.96,C -1.4618,E1 24.8862,E2 225.0895} C_DIS
LIN {X -85.8707,Y -88.5794,Z 130,A -137.2311,B 24.9597,C -1.4668,E1 24.8894,E2 223.4902} C_DIS
LIN {X -83.9668,Y -90.3887,Z 130,A -135.8711,B 24.9595,C -1.4706,E1 24.8922,E2 222.1154} C_DIS
LIN {X -81.4209,Y -92.6862,Z 130,A -134.4065,B 24.96,C -1.4616,E1 24.8952,E2 220.6665} C_DIS
LIN {X -79.1217,Y -94.6564,Z 130,A -133.1626,B 24.9605,C -1.4514,E1 24.8979,E2 219.4419} C_DIS
LIN {X -76.7749,Y -96.5697,Z 130,A -131.7282,B 24.9606,C -1.4501,E1 24.901,E2 218.0054} C_DIS
LIN {X -74.7028,Y -98.1836,Z 130,A -130.225,B 24.96,C -1.4608,E1 24.9044,E2 216.4711} C_DIS
LIN {X -71.944,Y -100.2205,Z 130,A -128.7592,B 24.9605,C -1.4522,E1 24.9076,E2 215.0206} C_DIS
LIN {X -69.4628,Y -101.9559,Z 130,A -127.3481,B 24.9606,C -1.4501,E1 24.9109,E2 213.6098} C_DIS
LIN {X -67.2776,Y -103.4131,Z 130,A -125.9911,B 24.9604,C -1.4545,E1 24.9141,E2 212.238} C_DIS
LIN {X -64.7194,Y -105.033,Z 130,A -124.5803,B 24.9604,C -1.4525,E1 24.9174,E2 210.8274} C_DIS
LIN {X -62.1223,Y -106.5897,Z 130,A -123.3023,B 24.9609,C -1.4445,E1 24.9205,E2 209.5646} C_DIS
LIN {X -59.4878,Y -108.0821,Z 130,A -121.7593,B 24.9607,C -1.4489,E1 24.9243,E2 208.0067} C_DIS
LIN {X -56.4599,Y -109.6922,Z 130,A -120.2949,B 24.9611,C -1.4409,E1 24.9279,E2 206.5573} C_DIS
LIN {X -54.1128,Y -110.8708,Z 130,A -119.0111,B 24.9611,C -1.4423,E1 24.9311,E2 205.2667} C_DIS
LIN {X -51.3756,Y -112.1654,Z 130,A -117.5294,B 24.9609,C -1.4442,E1 24.9349,E2 203.7768} C_DIS
LIN {X -48.2375,Y -113.5484,Z 130,A -116.2337,B 24.9618,C -1.4286,E1 24.9381,E2 202.5152} C_DIS
LIN {X -45.81,Y -114.5512,Z 130,A -114.7106,B 24.9611,C -1.4415,E1 24.9421,E2 200.958} C_DIS
LIN {X -42.6078,Y -115.7785,Z 130,A -113.2476,B 24.9615,C -1.434,E1 24.9459,E2 199.5098} C_DIS
LIN {X -39.7536,Y -116.7893,Z 130,A -111.8385,B 24.9615,C -1.4329,E1 24.9496,E2 198.1006} C_DIS
LIN {X -36.8755,Y -117.7297,Z 130,A -110.3738,B 24.9615,C -1.4346,E1 24.9536,E2 196.6293} C_DIS
LIN {X -32.5172,Y -119.0072,Z 130,A -108.3178,B 24.9617,C -1.4306,E1 24.9591,E2 194.5793} C_DIS
LIN {X -29.9553,Y -119.6795,Z 130,A -107.0952,B 24.9617,C -1.4295,E1 24.9624,E2 193.3576} C_DIS
LIN {X -27.0309,Y -120.3739,Z 130,A -105.5558,B 24.9614,C -1.4356,E1 24.9666,E2 191.8017} C_DIS
LIN {X -24.0686,Y -121.001,Z 130,A -104.1485,B 24.9614,C -1.4351,E1 24.9705,E2 190.394} C_DIS
LIN {X -21.0918,Y -121.5552,Z 130,A -102.8736,B 24.9618,C -1.4283,E1 24.9739,E2 189.1339} C_DIS
LIN {X -17.7049,Y -122.0927,Z 130,A -101.2801,B 24.9618,C -1.428,E1 24.9783,E2 187.5399} C_DIS
LIN {X -14.7848,Y -122.4809,Z 130,A -100.0445,B 24.9622,C -1.4214,E1 24.9817,E2 186.319} C_DIS
LIN {X -12.0925,Y -122.7775,Z 130,A -98.5207,B 24.9615,C -1.434,E1 24.986,E2 184.7645} C_DIS
LIN {X -9.0758,Y -123.0373,Z 130,A -97.1145,B 24.9615,C -1.434,E1 24.9899,E2 183.3577} C_DIS
LIN {X -6.0536,Y -123.2229,Z 130,A -95.8406,B 24.9618,C -1.4277,E1 24.9935,E2 182.0985} C_DIS
LIN {X -2.6263,Y -123.3418,Z 130,A -94.2333,B 24.9618,C -1.4286,E1 24.9979,E2 180.4886} C_DIS
LIN {X 0,Y -123.3715,Z 130,A -93.0291,B 24.9618,C -1.4281,E1 25.0013,E2 179.2857} C_DIS
LIN {X 0,Y -123.3715,Z 130,A -93.0291,B 24.9618,C -1.4281,E1 25.0013,E2 179.2857} C_DIS
Enddeposition()
LIN {X 0.8715,Y -122.5219,Z 130,A -93.0623,B 24.9621,C -1.422,E1 25.0012,E2 179.3333} C_DIS
Startdeposition()
$VEL.CP = VEL_PRINT
LIN {X -2.2553,Y -122.5043,Z 130,A -94.864,B 24.963,C -1.4056,E1 24.996,E2 181.1739} C_DIS
LIN {X -5.6128,Y -122.3969,Z 130,A -96.4036,B 24.963,C -1.4069,E1 24.9917,E2 182.7107} C_DIS
LIN {X -9.7069,Y -122.1399,Z 130,A -98.2578,B 24.9628,C -1.4099,E1 24.9866,E2 184.5585} C_DIS
LIN {X -13.1673,Y -121.8162,Z 130,A -99.9062,B 24.9628,C -1.409,E1 24.982,E2 186.21} C_DIS
LIN {X -16.1311,Y -121.4592,Z 130,A -101.2488,B 24.9627,C -1.4117,E1 24.9783,E2 187.5471} C_DIS
LIN {X -19.5381,Y -120.9591,Z 130,A -102.9627,B 24.9629,C -1.4073,E1 24.9735,E2 189.273} C_DIS
LIN {X -23.5094,Y -120.249,Z 130,A -104.7511,B 24.9626,C -1.4126,E1 24.9687,E2 191.0507} C_DIS
LIN {X -26.9713,Y -119.5212,Z 130,A -106.6374,B 24.9631,C -1.4026,E1 24.9634,E2 192.9631} C_DIS
LIN {X -30.6491,Y -118.6299,Z 130,A -108.2223,B 24.9626,C -1.4122,E1 24.9592,E2 194.5275} C_DIS
LIN {X -34.4852,Y -117.5725,Z 130,A -110.1917,B 24.9628,C -1.4084,E1 24.9539,E2 196.509} C_DIS
LIN {X -38.1599,Y -116.4321,Z 130,A -111.8533,B 24.9624,C -1.4161,E1 24.9495,E2 198.1552} C_DIS
LIN {X -41.0163,Y -115.4568,Z 130,A -113.2195,B 24.9623,C -1.4194,E1 24.9459,E2 199.5163} C_DIS
LIN {X -43.4121,Y -114.5765,Z 130,A -114.4836,B 24.9623,C -1.4173,E1 24.9426,E2 200.7881} C_DIS
LIN {X -47.0539,Y -113.1311,Z 130,A -116.3929,B 24.9625,C -1.4156,E1 24.9376,E2 202.7055} C_DIS
LIN {X -50.2081,Y -111.7656,Z 130,A -117.9587,B 24.9623,C -1.4193,E1 24.9336,E2 204.2663} C_DIS
LIN {X -53.3355,Y -110.3078,Z 130,A -119.5671,B 24.9621,C -1.4215,E1 24.9296,E2 205.8737} C_DIS
LIN {X -56.2394,Y -108.8568,Z 130,A -121.0353,B 24.9619,C -1.4257,E1 24.9259,E2 207.3358} C_DIS
LIN {X -58.8765,Y -107.4533,Z 130,A -122.5046,B 24.962,C -1.4243,E1 24.9223,E2 208.8127} C_DIS
LIN {X -62.4976,Y -105.3872,Z 130,A -124.5496,B 24.962,C -1.4228,E1 24.9173,E2 210.8673} C_DIS
LIN {X -65.8796,Y -103.3073,Z 130,A -126.4594,B 24.962,C -1.4232,E1 24.9128,E2 212.782} C_DIS
LIN {X -68.4051,Y -101.6526,Z 130,A -128.7141,B 24.9639,C -1.3879,E1 24.9074,E2 215.1281} C_DIS
LIN {X -73.5837,Y -97.9685,Z 130,A -130.5981,B 24.9611,C -1.4417,E1 24.9034,E2 216.8911} C_DIS
LIN {X -76.004,Y -96.103,Z 130,A -132.1143,B 24.9611,C -1.4404,E1 24.9001,E2 218.416} C_DIS
LIN {X -78.9052,Y -93.7384,Z 130,A -133.8491,B 24.9609,C -1.4444,E1 24.8963,E2 220.1479} C_DIS
LIN {X -80.6889,Y -92.2047,Z 130,A -134.9909,B 24.9609,C -1.4447,E1 24.8939,E2 221.2933} C_DIS
LIN {X -83.1933,Y -89.9527,Z 130,A -136.4963,B 24.9606,C -1.451,E1 24.8908,E2 222.7898} C_DIS
LIN {X -85.6926,Y -87.5757,Z 130,A -138.0931,B 24.9603,C -1.4551,E1 24.8876,E2 224.3835} C_DIS
LIN {X -88.5701,Y -84.6639,Z 130,A -140.1143,B 24.9603,C -1.4545,E1 24.8837,E2 226.4147} C_DIS
LIN {X -90.6723,Y -82.4091,Z 130,A -141.7028,B 24.9605,C -1.4512,E1 24.8806,E2 228.018} C_DIS
LIN {X -93.4236,Y -79.2747,Z 130,A -143.5448,B 24.96,C -1.4606,E1 24.8773,E2 229.8461} C_DIS
LIN {X -95.5676,Y -76.6784,Z 130,A -145.2852,B 24.9602,C -1.457,E1 24.8742,E2 231.6032} C_DIS
LIN {X -98.5047,Y -72.8668,Z 130,A -147.336,B 24.9594,C -1.4714,E1 24.8708,E2 233.6296} C_DIS
LIN {X -100.2416,Y -70.4586,Z 130,A -148.8937,B 24.9597,C -1.4674,E1 24.8682,E2 235.2043} C_DIS
LIN {X -102.5505,Y -67.0522,Z 130,A -150.6882,B 24.9591,C -1.4782,E1 24.8655,E2 236.9822} C_DIS
LIN {X -104.059,Y -64.6852,Z 130,A -152.0912,B 24.9591,C -1.4777,E1 24.8634,E2 238.3934} C_DIS
LIN {X -105.643,Y -62.0649,Z 130,A -153.4474,B 24.9587,C -1.4849,E1 24.8615,E2 239.7396} C_DIS
LIN {X -107.0773,Y -59.5557,Z 130,A -154.9032,B 24.9587,C -1.484,E1 24.8595,E2 241.2051} C_DIS
LIN {X -108.7416,Y -56.4639,Z 130,A -156.4453,B 24.9582,C -1.4929,E1 24.8575,E2 242.7341} C_DIS
LIN {X -109.9765,Y -54.0162,Z 130,A -157.8818,B 24.9584,C -1.4898,E1 24.8557,E2 244.1857} C_DIS
LIN {X -111.7231,Y -50.3024,Z 130,A -159.6954,B 24.9578,C -1.5,E1 24.8536,E2 245.985} C_DIS
LIN {X -113.1685,Y -46.9651,Z 130,A -161.3688,B 24.9575,C -1.5061,E1 24.8517,E2 247.6532} C_DIS
LIN {X -114.2701,Y -44.2168,Z 130,A -162.758,B 24.9573,C -1.51,E1 24.8503,E2 249.0408} C_DIS
LIN {X -116.0121,Y -39.4166,Z 130,A -165.0064,B 24.9565,C -1.5232,E1 24.8482,E2 251.2703} C_DIS
LIN {X -117.0207,Y -36.3118,Z 130,A -166.7834,B 24.9569,C -1.517,E1 24.8467,E2 253.0724} C_DIS
LIN {X -117.9716,Y -33.0937,Z 130,A -168.5237,B 24.957,C -1.5144,E1 24.8453,E2 254.8289} C_DIS
LIN {X -118.9998,Y -29.1799,Z 130,A -170.2645,B 24.9563,C -1.5269,E1 24.8441,E2 256.5502} C_DIS
LIN {X -119.704,Y -26.1409,Z 130,A -171.6895,B 24.956,C -1.5329,E1 24.8433,E2 257.9691} C_DIS
LIN {X -120.3812,Y -22.8226,Z 130,A -173.2816,B 24.9557,C -1.5376,E1 24.8424,E2 259.5596} C_DIS
LIN {X -121.0476,Y -18.9721,Z 130,A -175.1554,B 24.9555,C -1.5414,E1 24.8416,E2 261.4355} C_DIS
LIN {X -121.5877,Y -15.1389,Z 130,A -176.9098,B 24.955,C -1.5496,E1 24.8409,E2 263.1807} C_DIS
LIN {X -121.8774,Y -12.5828,Z 130,A -178.1199,B 24.9548,C -1.5532,E1 24.8405,E2 264.3895} C_DIS
LIN {X -122.1573,Y -9.4903,Z 130,A -179.6977,B 24.9548,C -1.5525,E1 24.8402,E2 265.9786} C_DIS
LIN {X -122.3865,Y -5.8544,Z 130,A 178.5876,B 24.9545,C -1.5575,E1 24.8399,E2 267.6916} C_DIS
LIN {X -122.5045,Y -2.2459,Z 130,A 176.9872,B 24.954,C -1.5668,E1 24.8398,E2 269.2793} C_DIS
LIN {X -122.5214,Y 0.9766,Z 130,A 175.4327,B 24.9538,C -1.5697,E1 24.8398,E2 270.8364} C_DIS
LIN {X -122.4266,Y 4.923,Z 130,A 173.5849,B 24.9535,C -1.5757,E1 24.84,E2 272.6811} C_DIS
LIN {X -122.2504,Y 8.1997,Z 130,A 171.983,B 24.9534,C -1.5778,E1 24.8402,E2 274.2875} C_DIS
LIN {X -121.9711,Y 11.6438,Z 130,A 170.433,B 24.9529,C -1.5859,E1 24.8406,E2 275.8275} C_DIS
LIN {X -121.5704,Y 15.2727,Z 130,A 168.6271,B 24.9528,C -1.5873,E1 24.8412,E2 277.641} C_DIS
LIN {X -121.037,Y 19.0405,Z 130,A 166.8053,B 24.9526,C -1.5913,E1 24.842,E2 279.4641} C_DIS
LIN {X -120.3376,Y 23.0491,Z 130,A 164.9665,B 24.952,C -1.6002,E1 24.8429,E2 281.2925} C_DIS
LIN {X -119.654,Y 26.3702,Z 130,A 163.2568,B 24.952,C -1.6,E1 24.8439,E2 283.0127} C_DIS
LIN {X -118.4658,Y 31.2844,Z 130,A 161.0689,B 24.9511,C -1.6152,E1 24.8453,E2 285.1773} C_DIS
LIN {X -117.3296,Y 35.3041,Z 130,A 159.0769,B 24.9508,C -1.6198,E1 24.8469,E2 287.1698} C_DIS
LIN {X -116.3282,Y 38.4791,Z 130,A 157.5198,B 24.9505,C -1.6247,E1 24.8482,E2 288.7242} C_DIS
LIN {X -115.5287,Y 40.8114,Z 130,A 156.2228,B 24.9507,C -1.6222,E1 24.8494,E2 290.0346} C_DIS
LIN {X -114.0494,Y 44.7785,Z 130,A 154.321,B 24.9501,C -1.6317,E1 24.8513,E2 291.9243} C_DIS
LIN {X -112.7104,Y 48.0523,Z 130,A 152.3968,B 24.9505,C -1.6252,E1 24.8534,E2 293.8747} C_DIS
LIN {X -110.7831,Y 52.3449,Z 130,A 150.3125,B 24.9498,C -1.6369,E1 24.8558,E2 295.9426} C_DIS
LIN {X -109.07,Y 55.8223,Z 130,A 148.5302,B 24.9494,C -1.6437,E1 24.858,E2 297.7182} C_DIS
LIN {X -107.3782,Y 59.0144,Z 130,A 146.9646,B 24.9487,C -1.654,E1 24.8601,E2 299.2675} C_DIS
LIN {X -105.997,Y 61.4593,Z 130,A 145.673,B 24.9484,C -1.6588,E1 24.8619,E2 300.5544} C_DIS
LIN {X -103.548,Y 65.5033,Z 130,A 143.4188,B 24.9482,C -1.6633,E1 24.8652,E2 302.8094} C_DIS
LIN {X -101.085,Y 69.2433,Z 130,A 141.1109,B 24.9484,C -1.66,E1 24.8688,E2 305.1368} C_DIS
LIN {X -98.7614,Y 72.5162,Z 130,A 139.2982,B 24.9479,C -1.668,E1 24.8717,E2 306.9393} C_DIS
LIN {X -96.0366,Y 76.088,Z 130,A 137.2232,B 24.9474,C -1.6748,E1 24.8753,E2 309.0079} C_DIS
LIN {X -94.1991,Y 78.3513,Z 130,A 135.8299,B 24.9473,C -1.6771,E1 24.8777,E2 310.4021} C_DIS
LIN {X -92.0254,Y 80.8941,Z 130,A 133.4846,B 24.9491,C -1.6474,E1 24.8822,E2 312.8287} C_DIS
LIN {X -88.2848,Y 84.9599,Z 130,A 131.7232,B 24.9465,C -1.6894,E1 24.8854,E2 314.4977} C_DIS
LIN {X -83.3852,Y 89.7766,Z 130,A 127.7603,B 24.9481,C -1.6645,E1 24.8936,E2 318.5362} C_DIS
LIN {X -79.6734,Y 93.0839,Z 130,A 126.3781,B 24.9451,C -1.711,E1 24.8963,E2 319.8132} C_DIS
LIN {X -77.5202,Y 94.8854,Z 130,A 124.7903,B 24.9457,C -1.7018,E1 24.8997,E2 321.4289} C_DIS
LIN {X -73.6254,Y 97.9371,Z 130,A 122.241,B 24.9461,C -1.6965,E1 24.9054,E2 324.0002} C_DIS
LIN {X -70.5806,Y 100.1563,Z 130,A 120.7496,B 24.9451,C -1.712,E1 24.9087,E2 325.4599} C_DIS
LIN {X -68.1199,Y 101.8457,Z 130,A 119.3672,B 24.9449,C -1.7154,E1 24.9119,E2 326.839} C_DIS
LIN {X -64.6634,Y 104.0726,Z 130,A 117.4404,B 24.9446,C -1.7189,E1 24.9165,E2 328.7634} C_DIS
LIN {X -61.8393,Y 105.7764,Z 130,A 115.3935,B 24.9459,C -1.6994,E1 24.9215,E2 330.8629} C_DIS
LIN {X -58.5808,Y 107.6137,Z 130,A 114.3693,B 24.9436,C -1.7346,E1 24.9238,E2 331.8063} C_DIS
LIN {X -56.7353,Y 108.5986,Z 130,A 113.1827,B 24.9441,C -1.727,E1 24.9268,E2 333.0144} C_DIS
LIN {X -53.7643,Y 110.1013,Z 130,A 111.5911,B 24.9441,C -1.728,E1 24.9308,E2 334.6078} C_DIS
LIN {X -51.1488,Y 111.3399,Z 130,A 109.9504,B 24.9447,C -1.7173,E1 24.935,E2 336.2781} C_DIS
LIN {X -47.2861,Y 113.0332,Z 130,A 108.1986,B 24.9439,C -1.73,E1 24.9394,E2 338.0037} C_DIS
LIN {X -42.8885,Y 114.7748,Z 130,A 105.8265,B 24.9442,C -1.7258,E1 24.9457,E2 340.3908} C_DIS
LIN {X -37.728,Y 116.5718,Z 130,A 103.4006,B 24.9436,C -1.7348,E1 24.952,E2 342.7999} C_DIS
LIN {X -33.9813,Y 117.7201,Z 130,A 101.4605,B 24.9438,C -1.732,E1 24.9573,E2 344.75} C_DIS
LIN {X -30.2857,Y 118.7233,Z 130,A 99.8369,B 24.9432,C -1.7414,E1 24.9616,E2 346.3537} C_DIS
LIN {X -27.2811,Y 119.4497,Z 130,A 98.2866,B 24.9434,C -1.738,E1 24.9658,E2 347.914} C_DIS
LIN {X -21.1949,Y 120.679,Z 130,A 95.5928,B 24.9426,C -1.7499,E1 24.9732,E2 350.5826} C_DIS
LIN {X -17.2862,Y 121.2995,Z 130,A 93.5688,B 24.943,C -1.7433,E1 24.9788,E2 352.6241} C_DIS
LIN {X -14.1073,Y 121.7103,Z 130,A 92.0629,B 24.943,C -1.7438,E1 24.9829,E2 354.1297} C_DIS
LIN {X -9.1833,Y 122.1818,Z 130,A 89.9011,B 24.9425,C -1.7519,E1 24.9889,E2 356.2735} C_DIS
LIN {X -3.772,Y 122.467,Z 130,A 87.2293,B 24.9428,C -1.7464,E1 24.9964,E2 358.9589} C_DIS
LIN {X -0.5036,Y 122.5243,Z 130,A 85.6454,B 24.943,C -1.7442,E1 25.0008,E2 360.548} C_DIS
LIN {X 3.4038,Y 122.4783,Z 130,A 83.6568,B 24.9435,C -1.7371,E1 25.0064,E2 362.5533} C_DIS
LIN {X 8.4056,Y 122.2365,Z 130,A 81.5987,B 24.9426,C -1.7502,E1 25.0121,E2 364.5795} C_DIS
LIN {X 11.2003,Y 122.0121,Z 130,A 80.2264,B 24.9428,C -1.7472,E1 25.0159,E2 365.958} C_DIS
LIN {X 14.6477,Y 121.647,Z 130,A 78.6558,B 24.9426,C -1.7493,E1 25.0203,E2 367.5226} C_DIS
LIN {X 17.781,Y 121.2292,Z 130,A 76.854,B 24.9437,C -1.7338,E1 25.0253,E2 369.3595} C_DIS
LIN {X 22.5006,Y 120.4432,Z 130,A 74.3822,B 24.9444,C -1.7221,E1 25.0322,E2 371.8564} C_DIS
LIN {X 26.4311,Y 119.6407,Z 130,A 73.0665,B 24.9428,C -1.7473,E1 25.0356,E2 373.1107} C_DIS
LIN {X 29.2473,Y 118.9833,Z 130,A 71.6297,B 24.9431,C -1.7426,E1 25.0396,E2 374.5567} C_DIS
LIN {X 33.0613,Y 117.9808,Z 130,A 69.8376,B 24.9431,C -1.7438,E1 25.0444,E2 376.343} C_DIS
LIN {X 36.2662,Y 117.0348,Z 130,A 68.21,B 24.9433,C -1.7395,E1 25.0487,E2 377.9778} C_DIS
LIN {X 39.4829,Y 115.9897,Z 130,A 66.7579,B 24.943,C -1.7443,E1 25.0525,E2 379.4158} C_DIS
LIN {X 42.0824,Y 115.0716,Z 130,A 65.315,B 24.9435,C -1.7359,E1 25.0564,E2 380.8758} C_DIS
LIN {X 46.2032,Y 113.4797,Z 130,A 63.2768,B 24.9435,C -1.7351,E1 25.0617,E2 382.9113} C_DIS
LIN {X 50.0719,Y 111.827,Z 130,A 61.2867,B 24.9438,C -1.7317,E1 25.0668,E2 384.9044} C_DIS
LIN {X 57.3332,Y 108.2837,Z 130,A 57.6416,B 24.9437,C -1.7332,E1 25.0759,E2 388.5361} C_DIS
LIN {X 60.4287,Y 106.5892,Z 130,A 55.8431,B 24.9443,C -1.7238,E1 25.0803,E2 390.3517} C_DIS
LIN {X 64.405,Y 104.2341,Z 130,A 53.9081,B 24.9438,C -1.7314,E1 25.0849,E2 392.2628} C_DIS
LIN {X 68.2191,Y 101.7785,Z 130,A 51.3967,B 24.9453,C -1.7092,E1 25.0908,E2 394.8184} C_DIS
LIN {X 72.4617,Y 98.8013,Z 130,A 49.3556,B 24.9443,C -1.7234,E1 25.0954,E2 396.8187} C_DIS
LIN {X 75.2248,Y 96.7157,Z 130,A 47.5731,B 24.945,C -1.7125,E1 25.0994,E2 398.6204} C_DIS
LIN {X 78.422,Y 94.1404,Z 130,A 45.7549,B 24.945,C -1.7138,E1 25.1033,E2 400.4288} C_DIS
LIN {X 80.9607,Y 91.9673,Z 130,A 44.2251,B 24.945,C -1.7122,E1 25.1065,E2 401.9561} C_DIS
LIN {X 83.0901,Y 90.0474,Z 130,A 42.942,B 24.945,C -1.7122,E1 25.1091,E2 403.234} C_DIS
LIN {X 85.4744,Y 87.789,Z 130,A 41.296,B 24.9456,C -1.7036,E1 25.1125,E2 404.8936} C_DIS
LIN {X 88.4465,Y 84.7922,Z 130,A 39.3028,B 24.9459,C -1.6984,E1 25.1164,E2 406.8907} C_DIS
LIN {X 90.7232,Y 82.3537,Z 130,A 37.8696,B 24.9458,C -1.701,E1 25.1191,E2 408.3113} C_DIS
LIN {X 92.76,Y 80.0531,Z 130,A 36.4244,B 24.946,C -1.6972,E1 25.1217,E2 409.7589} C_DIS
LIN {X 95.1633,Y 77.1773,Z 130,A 34.5854,B 24.9466,C -1.6888,E1 25.125,E2 411.6093} C_DIS
LIN {X 97.6756,Y 73.9736,Z 130,A 32.6806,B 24.9469,C -1.6841,E1 25.1283,E2 413.5163} C_DIS
LIN {X 99.8349,Y 71.031,Z 130,A 30.9424,B 24.9472,C -1.6782,E1 25.1311,E2 415.2599} C_DIS
LIN {X 102.2819,Y 67.4596,Z 130,A 29.0185,B 24.9472,C -1.6779,E1 25.1341,E2 417.175} C_DIS
LIN {X 104.2839,Y 64.3253,Z 130,A 27.2843,B 24.9475,C -1.6735,E1 25.1367,E2 418.9109} C_DIS
LIN {X 107.0339,Y 59.6335,Z 130,A 24.7738,B 24.9479,C -1.6682,E1 25.1402,E2 421.4209} C_DIS
LIN {X 108.589,Y 56.7536,Z 130,A 23.29,B 24.9479,C -1.6662,E1 25.1421,E2 422.9015} C_DIS
LIN {X 110.3108,Y 53.3291,Z 130,A 21.3963,B 24.9486,C -1.6561,E1 25.1445,E2 424.809} C_DIS
LIN {X 112.0425,Y 49.5918,Z 130,A 19.6282,B 24.9485,C -1.6583,E1 25.1465,E2 426.5622} C_DIS
LIN {X 113.2171,Y 46.8484,Z 130,A 18.233,B 24.9487,C -1.6542,E1 25.148,E2 427.9593} C_DIS
LIN {X 114.5044,Y 43.6026,Z 130,A 16.5402,B 24.9492,C -1.6464,E1 25.1498,E2 429.6612} C_DIS
LIN {X 115.6706,Y 40.4069,Z 130,A 14.9923,B 24.9494,C -1.6438,E1 25.1512,E2 431.2067} C_DIS
LIN {X 116.7413,Y 37.2042,Z 130,A 13.2965,B 24.95,C -1.6331,E1 25.1527,E2 432.9181} C_DIS
LIN {X 117.8205,Y 33.627,Z 130,A 11.6054,B 24.9502,C -1.6305,E1 25.154,E2 434.6056} C_DIS
LIN {X 118.8689,Y 29.7162,Z 130,A 9.8483,B 24.9502,C -1.6314,E1 25.1552,E2 436.3505} C_DIS
LIN {X 120.0114,Y 24.6914,Z 130,A 7.4132,B 24.9507,C -1.6226,E1 25.1567,E2 438.7922} C_DIS
LIN {X 120.6618,Y 21.2901,Z 130,A 5.7529,B 24.9511,C -1.6153,E1 25.1576,E2 440.4598} C_DIS
LIN {X 121.6082,Y 14.973,Z 130,A 2.6054,B 24.9522,C -1.5977,E1 25.1588,E2 443.6303} C_DIS
LIN {X 122.0565,Y 10.719,Z 130,A 0.8563,B 24.9518,C -1.6038,E1 25.1593,E2 445.3547} C_DIS
LIN {X 122.2814,Y 7.7405,Z 130,A -0.5675,B 24.9522,C -1.5979,E1 25.1595,E2 446.784} C_DIS
LIN {X 122.4766,Y 3.4585,Z 130,A -2.5929,B 24.9526,C -1.5903,E1 25.1598,E2 448.8152} C_DIS
LIN {X 122.5273,Y -0.0233,Z 130,A -4.1182,B 24.9526,C -1.5901,E1 25.1598,E2 450.3318} C_DIS
LIN {X 122.4565,Y -4.1134,Z 130,A -5.9781,B 24.9528,C -1.5865,E1 25.1597,E2 452.1891} C_DIS
LIN {X 122.3148,Y -7.1867,Z 130,A -7.5535,B 24.9535,C -1.5749,E1 25.1594,E2 453.7825} C_DIS
LIN {X 121.9365,Y -12.0176,Z 130,A -9.9065,B 24.9542,C -1.5631,E1 25.1589,E2 456.1496} C_DIS
LIN {X 121.433,Y -16.3331,Z 130,A -11.7115,B 24.9539,C -1.5678,E1 25.1582,E2 457.9327} C_DIS
LIN {X 120.9764,Y -19.4325,Z 130,A -13.266,B 24.9545,C -1.5585,E1 25.1576,E2 459.5} C_DIS
LIN {X 120.1727,Y -23.9047,Z 130,A -15.2812,B 24.9545,C -1.5571,E1 25.1566,E2 461.5067} C_DIS
LIN {X 119.5402,Y -26.889,Z 130,A -17.185,B 24.9562,C -1.5285,E1 25.1554,E2 463.4667} C_DIS
LIN {X 118.6796,Y -30.4557,Z 130,A -18.4111,B 24.9551,C -1.5476,E1 25.1546,E2 464.641} C_DIS
LIN {X 117.32,Y -35.3363,Z 130,A -20.7328,B 24.9554,C -1.5423,E1 25.1528,E2 466.9617} C_DIS
LIN {X 116.4666,Y -38.0531,Z 130,A -22.2397,B 24.9562,C -1.5293,E1 25.1515,E2 468.4909} C_DIS
LIN {X 114.5795,Y -43.4041,Z 130,A -24.4016,B 24.9552,C -1.5456,E1 25.1495,E2 470.602} C_DIS
LIN {X 113.2569,Y -46.7507,Z 130,A -26.4551,B 24.9566,C -1.5217,E1 25.1473,E2 472.7008} C_DIS
LIN {X 111.0535,Y -51.7639,Z 130,A -28.9356,B 24.9568,C -1.5178,E1 25.1445,E2 475.1768} C_DIS
LIN {X 109.6296,Y -54.7161,Z 130,A -30.4312,B 24.957,C -1.515,E1 25.1427,E2 476.6711} C_DIS
LIN {X 108.0603,Y -57.7575,Z 130,A -32.2649,B 24.9579,C -1.4985,E1 25.1402,E2 478.534} C_DIS
LIN {X 105.8383,Y -61.7345,Z 130,A -34.1479,B 24.9576,C -1.5045,E1 25.1377,E2 480.3929} C_DIS
LIN {X 104.2405,Y -64.3947,Z 130,A -35.8291,B 24.9585,C -1.4888,E1 25.1352,E2 482.1027} C_DIS
LIN {X 102.5385,Y -67.0704,Z 130,A -37.2826,B 24.9586,C -1.486,E1 25.133,E2 483.5555} C_DIS
LIN {X 99.118,Y -72.0292,Z 130,A -40.1163,B 24.9591,C -1.4773,E1 25.1284,E2 486.396} C_DIS
LIN {X 95.4804,Y -76.7861,Z 130,A -42.7833,B 24.9591,C -1.4763,E1 25.1239,E2 489.0527} C_DIS
LIN {X 93.1306,Y -79.6186,Z 130,A -44.3428,B 24.959,C -1.4798,E1 25.1211,E2 490.5969} C_DIS
LIN {X 91.032,Y -82.0104,Z 130,A -46.0542,B 24.9598,C -1.4648,E1 25.1178,E2 492.336} C_DIS
LIN {X 88.2081,Y -85.0396,Z 130,A -47.761,B 24.9594,C -1.4713,E1 25.1146,E2 494.02} C_DIS
LIN {X 86.0864,Y -87.1867,Z 130,A -49.1659,B 24.9596,C -1.4681,E1 25.1118,E2 495.4265} C_DIS
LIN {X 83.6688,Y -89.5101,Z 130,A -50.6991,B 24.9597,C -1.466,E1 25.1087,E2 496.9582} C_DIS
LIN {X 81.7285,Y -91.2844,Z 130,A -52.0202,B 24.9601,C -1.4586,E1 25.106,E2 498.2917} C_DIS
LIN {X 78.9756,Y -93.6784,Z 130,A -53.6211,B 24.9601,C -1.4598,E1 25.1026,E2 499.8834} C_DIS
LIN {X 75.4315,Y -96.5554,Z 130,A -55.7821,B 24.9604,C -1.4537,E1 25.0979,E2 502.0505} C_DIS
LIN {X 71.7192,Y -99.3439,Z 130,A -57.9323,B 24.9606,C -1.4501,E1 25.0931,E2 504.2016} C_DIS
LIN {X 67.7771,Y -102.0725,Z 130,A -60.0395,B 24.9605,C -1.4522,E1 25.0883,E2 506.2968} C_DIS
LIN {X 63.5726,Y -104.7422,Z 130,A -63.132,B 24.9627,C -1.4104,E1 25.0807,E2 509.4782} C_DIS
LIN {X 59.6977,Y -106.998,Z 130,A -64.596,B 24.9613,C -1.4374,E1 25.0773,E2 510.8741} C_DIS
LIN {X 56.8625,Y -108.5316,Z 130,A -66.1154,B 24.9615,C -1.4341,E1 25.0735,E2 512.3968} C_DIS
LIN {X 54.0559,Y -109.9568,Z 130,A -67.7051,B 24.9619,C -1.4259,E1 25.0695,E2 514.0016} C_DIS
LIN {X 49.7709,Y -111.9627,Z 130,A -70.2495,B 24.963,C -1.4064,E1 25.063,E2 516.5859} C_DIS
LIN {X 46.3689,Y -113.4123,Z 130,A -71.27,B 24.9613,C -1.4382,E1 25.0605,E2 517.5286} C_DIS
LIN {X 43.4392,Y -114.5663,Z 130,A -73.0054,B 24.962,C -1.4234,E1 25.0559,E2 519.2954} C_DIS
LIN {X 39.8163,Y -115.8773,Z 130,A -74.739,B 24.962,C -1.4243,E1 25.0514,E2 521.0234} C_DIS
LIN {X 36.0274,Y -117.1089,Z 130,A -76.631,B 24.9622,C -1.4206,E1 25.0463,E2 522.9205} C_DIS
LIN {X 33.3569,Y -117.897,Z 130,A -77.9533,B 24.9623,C -1.4182,E1 25.0428,E2 524.2464} C_DIS
LIN {X 29.6617,Y -118.8822,Z 130,A -79.7203,B 24.9623,C -1.4173,E1 25.038,E2 526.0127} C_DIS
LIN {X 25.0344,Y -119.9409,Z 130,A -81.7681,B 24.962,C -1.4235,E1 25.0325,E2 528.0431} C_DIS
LIN {X 19.2281,Y -121.008,Z 130,A -85.0717,B 24.9635,C -1.3953,E1 25.0232,E2 531.4099} C_DIS
LIN {X 15.9209,Y -121.4864,Z 130,A -86.4106,B 24.963,C -1.4049,E1 25.0196,E2 532.725} C_DIS
LIN {X 11.2179,Y -122.0104,Z 130,A -88.5099,B 24.9628,C -1.409,E1 25.0138,E2 534.813} C_DIS
LIN {X 7.8287,Y -122.2755,Z 130,A -90.0455,B 24.9628,C -1.4109,E1 25.0095,E2 536.3436} C_DIS
LIN {X 4.1785,Y -122.4545,Z 130,A -91.715,B 24.9626,C -1.4121,E1 25.0049,E2 538.0097} C_DIS
LIN {X 0.8715,Y -122.5219,Z 130,A -93.0605,B 24.9622,C -1.4212,E1 25.0012,E2 539.3333} C_DIS
Enddeposition()
LIN {X 0.8715,Y -122.5219,Z 130,A -93.0605,B 24.9622,C -1.4212,E1 25.0012,E2 539.3333} C_DIS
Startdeposition()
$VEL.CP = VEL_PRINT
LIN {X 3.9867,Y -121.6158,Z 130,A -91.1685,B 24.9603,C -1.4566,E1 25.0067,E2 537.3579} C_DIS
LIN {X 9.6625,Y -121.2966,Z 130,A -88.5075,B 24.9603,C -1.457,E1 25.0141,E2 534.697} C_DIS
LIN {X 13.3965,Y -120.9434,Z 130,A -86.1228,B 24.9585,C -1.4878,E1 25.0209,E2 532.241} C_DIS
LIN {X 17.9228,Y -120.3556,Z 130,A -84.6593,B 24.9603,C -1.4562,E1 25.0248,E2 530.8537} C_DIS
LIN {X 20.5423,Y -119.9353,Z 130,A -82.8024,B 24.9586,C -1.4865,E1 25.0301,E2 528.9269} C_DIS
LIN {X 24.6598,Y -119.1561,Z 130,A -81.4044,B 24.96,C -1.4604,E1 25.0337,E2 527.5925} C_DIS
LIN {X 27.1499,Y -118.6136,Z 130,A -80.0301,B 24.9595,C -1.47,E1 25.0375,E2 526.1974} C_DIS
LIN {X 31.2628,Y -117.5973,Z 130,A -78.1182,B 24.9596,C -1.468,E1 25.0427,E2 524.2931} C_DIS
LIN {X 34.5873,Y -116.6617,Z 130,A -76.6325,B 24.9599,C -1.463,E1 25.0466,E2 522.8216} C_DIS
LIN {X 42.0944,Y -114.1687,Z 130,A -72.7859,B 24.9593,C -1.4736,E1 25.0568,E2 518.9575} C_DIS
LIN {X 45.5255,Y -112.8442,Z 130,A -71.1202,B 24.9593,C -1.4729,E1 25.0611,E2 517.2973} C_DIS
LIN {X 51.89,Y -110.0637,Z 130,A -67.8106,B 24.959,C -1.4798,E1 25.0696,E2 513.9796} C_DIS
LIN {X 54.9984,Y -108.5431,Z 130,A -66.1789,B 24.9588,C -1.4826,E1 25.0737,E2 512.3455} C_DIS
LIN {X 57.549,Y -107.213,Z 130,A -64.7765,B 24.9586,C -1.4873,E1 25.0772,E2 510.936} C_DIS
LIN {X 65.352,Y -102.6429,Z 130,A -60.4895,B 24.958,C -1.4967,E1 25.0875,E2 506.6401} C_DIS
LIN {X 68.079,Y -100.854,Z 130,A -58.6778,B 24.9571,C -1.5135,E1 25.0917,E2 504.7948} C_DIS
LIN {X 71.2676,Y -98.6291,Z 130,A -57.3348,B 24.9582,C -1.4931,E1 25.0946,E2 503.5048} C_DIS
LIN {X 73.8309,Y -96.7241,Z 130,A -55.7255,B 24.9578,C -1.5016,E1 25.0983,E2 501.8813} C_DIS
LIN {X 76.6654,Y -94.4915,Z 130,A -54.1917,B 24.958,C -1.4972,E1 25.1016,E2 500.3637} C_DIS
LIN {X 80.5173,Y -91.2337,Z 130,A -51.4058,B 24.9565,C -1.5231,E1 25.1076,E2 497.5275} C_DIS
LIN {X 82.9305,Y -89.0456,Z 130,A -50.1713,B 24.9572,C -1.5118,E1 25.11,E2 496.3246} C_DIS
LIN {X 85.4658,Y -86.6132,Z 130,A -48.5583,B 24.9571,C -1.5138,E1 25.1133,E2 494.7136} C_DIS
LIN {X 89.4634,Y -82.478,Z 130,A -45.2369,B 24.9549,C -1.5515,E1 25.1198,E2 491.3177} C_DIS
LIN {X 92.5799,Y -78.9633,Z 130,A -43.6991,B 24.9565,C -1.5234,E1 25.1224,E2 489.8533} C_DIS
LIN {X 94.64,Y -76.4823,Z 130,A -41.5002,B 24.9543,C -1.5617,E1 25.1264,E2 487.574} C_DIS
LIN {X 97.6505,Y -72.6015,Z 130,A -39.9312,B 24.9561,C -1.5305,E1 25.1289,E2 486.0861} C_DIS
LIN {X 101.0699,Y -67.76,Z 130,A -36.9824,B 24.9552,C -1.5463,E1 25.1337,E2 483.1146} C_DIS
LIN {X 103.1614,Y -64.5288,Z 130,A -35.215,B 24.955,C -1.5493,E1 25.1363,E2 481.3491} C_DIS
LIN {X 105.3606,Y -60.8725,Z 130,A -33.5265,B 24.9556,C -1.5391,E1 25.1387,E2 479.6934} C_DIS
LIN {X 107.2406,Y -57.4981,Z 130,A -31.3658,B 24.9543,C -1.5617,E1 25.1416,E2 477.4907} C_DIS
LIN {X 108.8824,Y -54.3227,Z 130,A -29.7968,B 24.9543,C -1.561,E1 25.1436,E2 475.9316} C_DIS
LIN {X 110.111,Y -51.7883,Z 130,A -27.3532,B 24.9507,C -1.622,E1 25.1467,E2 473.3574} C_DIS
LIN {X 112.9647,Y -45.2295,Z 130,A -24.2243,B 24.9508,C -1.6202,E1 25.1498,E2 470.2501} C_DIS
LIN {X 115.0831,Y -39.5296,Z 130,A -22.232,B 24.9529,C -1.5848,E1 25.1516,E2 468.3524} C_DIS
LIN {X 116.1646,Y -36.2225,Z 130,A -20.7358,B 24.9531,C -1.5828,E1 25.1529,E2 466.8692} C_DIS
LIN {X 117.083,Y -33.1332,Z 130,A -19.1798,B 24.9527,C -1.5897,E1 25.1541,E2 465.3061} C_DIS
LIN {X 117.9319,Y -29.9737,Z 130,A -17.5451,B 24.9521,C -1.5994,E1 25.1552,E2 463.6578} C_DIS
LIN {X 118.8656,Y -26.0231,Z 130,A -15.7598,B 24.9521,C -1.5992,E1 25.1563,E2 461.8833} C_DIS
LIN {X 119.5585,Y -22.6307,Z 130,A -13.896,B 24.951,C -1.6163,E1 25.1573,E2 459.9901} C_DIS
LIN {X 120.3926,Y -17.6684,Z 130,A -11.7631,B 24.9513,C -1.6121,E1 25.1583,E2 457.8797} C_DIS
LIN {X 120.8171,Y -14.4766,Z 130,A -10.2812,B 24.9511,C -1.6153,E1 25.1588,E2 456.3989} C_DIS
LIN {X 121.3922,Y -8.3786,Z 130,A -7.4248,B 24.9506,C -1.6234,E1 25.1595,E2 453.5405} C_DIS
LIN {X 121.5511,Y -5.6343,Z 130,A -5.504,B 24.9484,C -1.6594,E1 25.1597,E2 451.5461} C_DIS
LIN {X 121.6767,Y -1.0651,Z 130,A -4.0818,B 24.9503,C -1.6294,E1 25.1598,E2 450.2032} C_DIS
LIN {X 121.6064,Y 4.2955,Z 130,A -0.9109,B 24.9477,C -1.6704,E1 25.1596,E2 446.9544} C_DIS
LIN {X 121.3781,Y 8.5869,Z 130,A 0.6683,B 24.9487,C -1.6544,E1 25.1593,E2 445.4223} C_DIS
LIN {X 121.1142,Y 11.7431,Z 130,A 2.6376,B 24.9469,C -1.6835,E1 25.1587,E2 443.3961} C_DIS
LIN {X 120.5763,Y 16.3751,Z 130,A 4.4972,B 24.9475,C -1.6735,E1 25.1581,E2 441.5712} C_DIS
LIN {X 119.5767,Y 22.5363,Z 130,A 7.1896,B 24.9477,C -1.6704,E1 25.1568,E2 438.9019} C_DIS
LIN {X 118.3609,Y 28.237,Z 130,A 9.9543,B 24.9471,C -1.68,E1 25.1551,E2 436.1305} C_DIS
LIN {X 117.4567,Y 31.7832,Z 130,A 11.532,B 24.9472,C -1.6781,E1 25.154,E2 434.5664} C_DIS
LIN {X 116.538,Y 35.0043,Z 130,A 13.2539,B 24.9465,C -1.6902,E1 25.1526,E2 432.8257} C_DIS
LIN {X 115.3649,Y 38.6938,Z 130,A 14.9471,B 24.9465,C -1.6893,E1 25.1511,E2 431.1444} C_DIS
LIN {X 114.2629,Y 41.836,Z 130,A 16.6753,B 24.9457,C -1.702,E1 25.1495,E2 429.3958} C_DIS
LIN {X 112.7301,Y 45.8057,Z 130,A 18.4311,B 24.9461,C -1.6955,E1 25.1477,E2 427.665} C_DIS
LIN {X 110.7825,Y 50.3351,Z 130,A 20.9226,B 24.9452,C -1.7108,E1 25.1449,E2 425.1512} C_DIS
LIN {X 109.1011,Y 53.8816,Z 130,A 22.626,B 24.9452,C -1.7088,E1 25.1428,E2 423.4615} C_DIS
LIN {X 107.6685,Y 56.6898,Z 130,A 24.118,B 24.945,C -1.7134,E1 25.1409,E2 421.9666} C_DIS
LIN {X 106.1814,Y 59.4287,Z 130,A 26.7688,B 24.9408,C -1.7769,E1 25.1371,E2 419.1796} C_DIS
LIN {X 102.3763,Y 65.7673,Z 130,A 28.6815,B 24.9454,C -1.7076,E1 25.1345,E2 417.4403} C_DIS
LIN {X 99.952,Y 69.3963,Z 130,A 31.0513,B 24.944,C -1.7285,E1 25.1308,E2 415.033} C_DIS
LIN {X 98.0812,Y 72.0163,Z 130,A 32.6231,B 24.9436,C -1.7351,E1 25.1282,E2 413.4532} C_DIS
LIN {X 95.6934,Y 75.1608,Z 130,A 34.4541,B 24.9434,C -1.7383,E1 25.125,E2 411.6234} C_DIS
LIN {X 93.4282,Y 77.9582,Z 130,A 36.1516,B 24.9431,C -1.7425,E1 25.122,E2 409.9237} C_DIS
LIN {X 90.817,Y 80.985,Z 130,A 37.9,B 24.9432,C -1.7402,E1 25.1188,E2 408.1884} C_DIS
LIN {X 88.9796,Y 83.0007,Z 130,A 39.3265,B 24.9426,C -1.7501,E1 25.1161,E2 406.7448} C_DIS
LIN {X 86.9317,Y 85.1434,Z 130,A 40.7196,B 24.9424,C -1.7531,E1 25.1134,E2 405.3508} C_DIS
LIN {X 84.4485,Y 87.6053,Z 130,A 42.2661,B 24.9424,C -1.7517,E1 25.1103,E2 403.8139} C_DIS
LIN {X 82.664,Y 89.2927,Z 130,A 43.8079,B 24.9411,C -1.773,E1 25.1071,E2 402.2282} C_DIS
LIN {X 80.1982,Y 91.5125,Z 130,A 45.013,B 24.942,C -1.7587,E1 25.1046,E2 401.0617} C_DIS
LIN {X 77.6298,Y 93.7011,Z 130,A 46.5914,B 24.9419,C -1.7612,E1 25.1012,E2 399.4833} C_DIS
LIN {X 74.5341,Y 96.1822,Z 130,A 48.4714,B 24.9416,C -1.7653,E1 25.0971,E2 397.6007} C_DIS
LIN {X 71.755,Y 98.2725,Z 130,A 50.0533,B 24.9416,C -1.7655,E1 25.0936,E2 396.0239} C_DIS
LIN {X 65.0517,Y 102.8348,Z 130,A 54.4527,B 24.9393,C -1.8,E1 25.0832,E2 391.5577} C_DIS
LIN {X 61.2991,Y 105.115,Z 130,A 56.0163,B 24.9407,C -1.7786,E1 25.0796,E2 390.0495} C_DIS
LIN {X 58.1294,Y 106.8982,Z 130,A 57.6603,B 24.9407,C -1.7777,E1 25.0755,E2 388.4123} C_DIS
LIN {X 53.7459,Y 109.1684,Z 130,A 60.2842,B 24.9396,C -1.7952,E1 25.0689,E2 385.7543} C_DIS
LIN {X 50.8139,Y 110.5646,Z 130,A 61.5746,B 24.9402,C -1.7855,E1 25.0657,E2 384.4901} C_DIS
LIN {X 48.2131,Y 111.7226,Z 130,A 62.8684,B 24.9402,C -1.7848,E1 25.0624,E2 383.2011} C_DIS
LIN {X 44.7512,Y 113.1532,Z 130,A 64.3554,B 24.9411,C -1.7734,E1 25.0586,E2 381.7444} C_DIS
LIN {X 42.1842,Y 114.1359,Z 130,A 65.9717,B 24.9399,C -1.79,E1 25.0543,E2 380.0923} C_DIS
LIN {X 38.8317,Y 115.3184,Z 130,A 67.5514,B 24.9401,C -1.787,E1 25.0502,E2 378.5229} C_DIS
LIN {X 35.191,Y 116.4826,Z 130,A 69.4187,B 24.9398,C -1.7916,E1 25.0452,E2 376.648} C_DIS
LIN {X 31.7743,Y 117.4591,Z 130,A 71.0131,B 24.94,C -1.789,E1 25.0409,E2 375.0623} C_DIS
LIN {X 28.106,Y 118.3927,Z 130,A 72.9129,B 24.9396,C -1.7956,E1 25.0357,E2 373.1497} C_DIS
LIN {X 22.4964,Y 119.5842,Z 130,A 75.6187,B 24.9395,C -1.7971,E1 25.0283,E2 370.4437} C_DIS
LIN {X 19.7313,Y 120.0709,Z 130,A 77.1179,B 24.9389,C -1.8059,E1 25.0242,E2 368.9252} C_DIS
LIN {X 14.9356,Y 120.7629,Z 130,A 79.385,B 24.9389,C -1.8057,E1 25.0179,E2 366.6604} C_DIS
LIN {X 9.8909,Y 121.2784,Z 130,A 81.2791,B 24.9404,C -1.7829,E1 25.0128,E2 364.8215} C_DIS
LIN {X 4.3782,Y 121.603,Z 130,A 84.0104,B 24.94,C -1.7889,E1 25.0051,E2 362.077} C_DIS
LIN {X -1.0065,Y 121.677,Z 130,A 86.6436,B 24.9397,C -1.7929,E1 24.9977,E2 359.4343} C_DIS
LIN {X -8.5276,Y 121.3821,Z 130,A 89.9621,B 24.9405,C -1.7812,E1 24.9886,E2 356.1429} C_DIS
LIN {X -15.75,Y 120.6573,Z 130,A 93.2775,B 24.941,C -1.7746,E1 24.9794,E2 352.8411} C_DIS
LIN {X -24.9395,Y 119.0986,Z 130,A 98.1132,B 24.9398,C -1.7915,E1 24.966,E2 347.9606} C_DIS
LIN {X -28.5851,Y 118.276,Z 130,A 99.7815,B 24.9402,C -1.7857,E1 24.9615,E2 346.304} C_DIS
LIN {X -31.6627,Y 117.4892,Z 130,A 101.2066,B 24.9406,C -1.781,E1 24.9576,E2 344.8879} C_DIS
LIN {X -34.6798,Y 116.6343,Z 130,A 102.7409,B 24.9405,C -1.7819,E1 24.9535,E2 343.3488} C_DIS
LIN {X -37.7032,Y 115.6926,Z 130,A 104.7911,B 24.9389,C -1.8056,E1 24.9479,E2 341.2387} C_DIS
LIN {X -41.7703,Y 114.2869,Z 130,A 106.0167,B 24.9415,C -1.7667,E1 24.9449,E2 340.1031} C_DIS
LIN {X -45.1984,Y 112.9773,Z 130,A 108.1318,B 24.9405,C -1.7817,E1 24.9393,E2 337.9477} C_DIS
LIN {X -48.401,Y 111.6407,Z 130,A 109.5968,B 24.9412,C -1.7717,E1 24.9356,E2 336.503} C_DIS
LIN {X -51.4542,Y 110.2666,Z 130,A 111.2601,B 24.9411,C -1.7732,E1 24.9313,E2 334.8322} C_DIS
LIN {X -55.0386,Y 108.5225,Z 130,A 113.146,B 24.9412,C -1.7705,E1 24.9266,E2 332.9476} C_DIS
LIN {X -58.0266,Y 106.954,Z 130,A 115.4618,B 24.9392,C -1.8005,E1 24.9208,E2 330.5539} C_DIS
LIN {X -62.6651,Y 104.3055,Z 130,A 117.2697,B 24.9417,C -1.7641,E1 24.9166,E2 328.8272} C_DIS
LIN {X -66.7601,Y 101.732,Z 130,A 119.5293,B 24.942,C -1.7589,E1 24.9113,E2 326.5728} C_DIS
LIN {X -69.1089,Y 100.1518,Z 130,A 120.9895,B 24.9418,C -1.7619,E1 24.9079,E2 325.1006} C_DIS
LIN {X -71.5364,Y 98.4325,Z 130,A 122.3429,B 24.9422,C -1.7569,E1 24.9049,E2 323.7543} C_DIS
LIN {X -74.9281,Y 95.8773,Z 130,A 124.1868,B 24.9429,C -1.7456,E1 24.9008,E2 321.9304} C_DIS
LIN {X -78.3917,Y 93.0669,Z 130,A 126.4677,B 24.9427,C -1.7489,E1 24.8959,E2 319.6331} C_DIS
LIN {X -82.7955,Y 89.172,Z 130,A 129.6918,B 24.9418,C -1.7627,E1 24.8891,E2 316.3633} C_DIS
LIN {X -85.755,Y 86.3275,Z 130,A 131.2272,B 24.9432,C -1.7404,E1 24.8862,E2 314.8745} C_DIS
LIN {X -88.5202,Y 83.4892,Z 130,A 133.5077,B 24.9423,C -1.754,E1 24.8817,E2 312.5516} C_DIS
LIN {X -91.3647,Y 80.3674,Z 130,A 134.9697,B 24.9442,C -1.7256,E1 24.8791,E2 311.1505} C_DIS
LIN {X -93.4751,Y 77.9017,Z 130,A 136.6838,B 24.9439,C -1.7298,E1 24.876,E2 309.4187} C_DIS
LIN {X -95.8354,Y 74.9811,Z 130,A 138.5706,B 24.9439,C -1.7302,E1 24.8727,E2 307.5221} C_DIS
LIN {X -98.7987,Y 71.0299,Z 130,A 140.6573,B 24.945,C -1.7134,E1 24.8693,E2 305.4655} C_DIS
LIN {X -101.4914,Y 67.125,Z 130,A 142.8733,B 24.9454,C -1.7063,E1 24.8658,E2 303.2552} C_DIS
LIN {X -103.8551,Y 63.4068,Z 130,A 145.0923,B 24.9454,C -1.7066,E1 24.8625,E2 301.0241} C_DIS
LIN {X -107.0895,Y 57.7767,Z 130,A 148.0983,B 24.9461,C -1.6953,E1 24.8585,E2 298.0293} C_DIS
LIN {X -109.0184,Y 54.0484,Z 130,A 149.9789,B 24.9468,C -1.6852,E1 24.8561,E2 296.1627} C_DIS
LIN {X -111.8571,Y 47.9032,Z 130,A 153.3537,B 24.9468,C -1.6835,E1 24.8522,E2 292.7735} C_DIS
LIN {X -113.2018,Y 44.6276,Z 130,A 154.8532,B 24.9477,C -1.6711,E1 24.8506,E2 291.2952} C_DIS
LIN {X -114.8818,Y 40.1055,Z 130,A 157.2192,B 24.9479,C -1.6681,E1 24.8484,E2 288.9231} C_DIS
LIN {X -116.0753,Y 36.5103,Z 130,A 158.9209,B 24.9484,C -1.6588,E1 24.8469,E2 287.2336} C_DIS
LIN {X -117.2271,Y 32.6245,Z 130,A 161.5292,B 24.9469,C -1.6832,E1 24.8449,E2 284.5522} C_DIS
LIN {X -118.3648,Y 28.221,Z 130,A 163.2061,B 24.9486,C -1.656,E1 24.8438,E2 282.9303} C_DIS
LIN {X -119.1544,Y 24.668,Z 130,A 164.8405,B 24.9492,C -1.647,E1 24.8429,E2 281.3076} C_DIS
LIN {X -119.8837,Y 20.848,Z 130,A 166.6913,B 24.9495,C -1.6419,E1 24.8419,E2 279.4581} C_DIS
LIN {X -120.4456,Y 17.2954,Z 130,A 168.3037,B 24.95,C -1.6329,E1 24.8413,E2 277.8576} C_DIS
LIN {X -120.8684,Y 14.0388,Z 130,A 169.9355,B 24.9501,C -1.6315,E1 24.8407,E2 276.2193} C_DIS
LIN {X -121.2558,Y 10.173,Z 130,A 171.8196,B 24.9503,C -1.6279,E1 24.8402,E2 274.3325} C_DIS
LIN {X -121.5044,Y 6.5527,Z 130,A 173.496,B 24.9508,C -1.6209,E1 24.84,E2 272.6627} C_DIS
LIN {X -121.6526,Y 2.6548,Z 130,A 175.3732,B 24.951,C -1.6166,E1 24.8398,E2 270.7844} C_DIS
LIN {X -121.679,Y -0.6946,Z 130,A 176.8847,B 24.9515,C -1.6086,E1 24.8398,E2 269.2828} C_DIS
LIN {X -121.6184,Y -3.9042,Z 130,A 178.4855,B 24.9515,C -1.6076,E1 24.8399,E2 267.6749} C_DIS
LIN {X -121.4224,Y -7.9323,Z 130,A -179.6813,B 24.9521,C -1.5985,E1 24.8402,E2 265.8522} C_DIS
LIN {X -121.1796,Y -11.0344,Z 130,A -178.1831,B 24.9523,C -1.5952,E1 24.8406,E2 264.3528} C_DIS
LIN {X -120.854,Y -14.1616,Z 130,A -176.6819,B 24.9525,C -1.5914,E1 24.841,E2 262.8519} C_DIS
LIN {X -120.3583,Y -17.9044,Z 130,A -174.7905,B 24.9525,C -1.5906,E1 24.8418,E2 260.9512} C_DIS
LIN {X -119.81,Y -21.2575,Z 130,A -173.2682,B 24.9531,C -1.5821,E1 24.8425,E2 259.4399} C_DIS
LIN {X -119.2364,Y -24.2688,Z 130,A -171.8151,B 24.9533,C -1.578,E1 24.8433,E2 257.9881} C_DIS
LIN {X -118.564,Y -27.3647,Z 130,A -170.3132,B 24.9536,C -1.5737,E1 24.8442,E2 256.4874} C_DIS
LIN {X -117.88,Y -30.1753,Z 130,A -168.2959,B 24.9521,C -1.5982,E1 24.8457,E2 254.4} C_DIS
LIN {X -116.5972,Y -34.8048,Z 130,A -166.6372,B 24.9541,C -1.5647,E1 24.8469,E2 252.8116} C_DIS
LIN {X -115.3631,Y -38.6991,Z 130,A -164.6072,B 24.9541,C -1.5635,E1 24.8487,E2 250.7729} C_DIS
LIN {X -113.4597,Y -43.971,Z 130,A -162.0678,B 24.9549,C -1.5513,E1 24.8511,E2 248.2484} C_DIS
LIN {X -112.075,Y -47.3862,Z 130,A -160.3373,B 24.9552,C -1.546,E1 24.853,E2 246.5209} C_DIS
LIN {X -110.485,Y -50.9849,Z 130,A -158.506,B 24.9556,C -1.5397,E1 24.8551,E2 244.6945} C_DIS
LIN {X -109.0822,Y -53.9196,Z 130,A -156.9339,B 24.9557,C -1.5371,E1 24.857,E2 243.1201} C_DIS
LIN {X -107.2851,Y -57.4162,Z 130,A -154.9598,B 24.9557,C -1.5373,E1 24.8596,E2 241.1349} C_DIS
LIN {X -105.4258,Y -60.7591,Z 130,A -152.9172,B 24.9554,C -1.5431,E1 24.8624,E2 239.0679} C_DIS
LIN {X -103.6861,Y -63.6849,Z 130,A -151.5339,B 24.9562,C -1.5291,E1 24.8644,E2 237.7109} C_DIS
LIN {X -101.1893,Y -67.583,Z 130,A -149.4235,B 24.9567,C -1.5203,E1 24.8676,E2 235.6109} C_DIS
LIN {X -99.2569,Y -70.3877,Z 130,A -147.7917,B 24.9569,C -1.5175,E1 24.8702,E2 233.9778} C_DIS
LIN {X -96.8949,Y -73.6074,Z 130,A -145.6363,B 24.9564,C -1.525,E1 24.8739,E2 231.7939} C_DIS
LIN {X -93.7068,Y -77.6229,Z 130,A -143.5758,B 24.9577,C -1.5035,E1 24.8774,E2 229.7751} C_DIS
LIN {X -92.062,Y -79.569,Z 130,A -141.8937,B 24.9566,C -1.5222,E1 24.8806,E2 228.0408} C_DIS
LIN {X -89.6668,Y -82.2563,Z 130,A -140.5996,B 24.9578,C -1.5004,E1 24.8829,E2 226.7928} C_DIS
LIN {X -86.8116,Y -85.2649,Z 130,A -138.8699,B 24.9586,C -1.4861,E1 24.8862,E2 225.0897} C_DIS
LIN {X -83.4199,Y -88.5853,Z 130,A -136.4047,B 24.9583,C -1.4917,E1 24.8912,E2 222.601} C_DIS
LIN {X -80.7619,Y -91.0167,Z 130,A -134.6032,B 24.9583,C -1.493,E1 24.895,E2 220.7893} C_DIS
LIN {X -78.2849,Y -93.1567,Z 130,A -133.0518,B 24.9583,C -1.4904,E1 24.8983,E2 219.2379} C_DIS
LIN {X -75.233,Y -95.6363,Z 130,A -131.3233,B 24.9589,C -1.4814,E1 24.902,E2 217.5244} C_DIS
LIN {X -73.3541,Y -97.0851,Z 130,A -129.396,B 24.9569,C -1.5163,E1 24.9066,E2 215.5071} C_DIS
LIN {X -68.9574,Y -100.2569,Z 130,A -127.5521,B 24.959,C -1.4796,E1 24.9106,E2 213.7444} C_DIS
LIN {X -65.81,Y -102.3489,Z 130,A -125.7259,B 24.959,C -1.4789,E1 24.9149,E2 211.9139} C_DIS
LIN {X -62.1839,Y -104.5921,Z 130,A -123.8783,B 24.9596,C -1.4685,E1 24.9192,E2 210.0851} C_DIS
LIN {X -59.5704,Y -106.1022,Z 130,A -122.435,B 24.9596,C -1.4675,E1 24.9227,E2 208.64} C_DIS
LIN {X -57.0151,Y -107.4972,Z 130,A -121.0112,B 24.9596,C -1.4681,E1 24.9262,E2 207.2108} C_DIS
LIN {X -54.0323,Y -109.0264,Z 130,A -119.4022,B 24.9596,C -1.4675,E1 24.9303,E2 205.5989} C_DIS
LIN {X -50.7267,Y -110.6052,Z 130,A -117.5085,B 24.9593,C -1.4732,E1 24.9351,E2 203.6869} C_DIS
LIN {X -46.8955,Y -112.2818,Z 130,A -115.5769,B 24.9596,C -1.4694,E1 24.9401,E2 201.7599} C_DIS
Enddeposition()
END
